SPLINE
SPL {X  -165.650, Y  +484.445, Z    +0.000, E1   +32.277, E3 +483766.169}
SPL {X  -165.650, Y  +481.524, Z    +0.000, E1   +31.089, E3 +483783.620}
SPL {X  -165.650, Y  +478.014, Z    +0.000, E1   +30.826, E3 +483797.227}
SPL {X  -165.650, Y  +474.473, Z    +0.000, E1   +30.943, E3 +483808.552}
SPL {X  -165.650, Y  +470.376, Z    +0.000, E1   +30.888, E3 +483823.081}
SPL {X  -165.650, Y  +465.146, Z    +0.000, E1   +30.883, E3 +483841.012}
SPL {X  -165.650, Y  +461.106, Z    +0.000, E1   +30.916, E3 +483854.430}
SPL {X  -165.650, Y  +458.435, Z    +0.000, E1   +30.759, E3 +483864.638}
SPL {X  -165.650, Y  +454.220, Z    +0.000, E1   +30.954, E3 +483877.871}
SPL {X  -165.650, Y  +450.433, Z    +0.000, E1   +30.789, E3 +483891.835}
SPL {X  -165.650, Y  +447.097, Z    +0.000, E1   +30.843, E3 +483902.884}
SPL {X  -165.650, Y  +443.673, Z    +0.000, E1   +30.907, E3 +483914.192}
SPL {X  -165.650, Y  +440.976, Z    +0.000, E1   +30.719, E3 +483924.648}
SPL {X  -165.650, Y  +436.324, Z    +0.000, E1   +30.994, E3 +483938.935}
SPL {X  -165.650, Y  +432.765, Z    +0.000, E1   +30.831, E3 +483951.935}
SPL {X  -165.650, Y  +429.309, Z    +0.000, E1   +30.920, E3 +483963.276}
SPL {X  -165.650, Y  +424.918, Z    +0.000, E1   +30.862, E3 +483978.733}
SPL {X  -165.650, Y  +421.437, Z    +0.000, E1   +30.833, E3 +483990.701}
SPL {X  -165.650, Y  +418.489, Z    +0.000, E1   +30.835, E3 +484000.818}
SPL {X  -165.650, Y  +414.127, Z    +0.000, E1   +30.869, E3 +484015.726}
SPL {X  -165.650, Y  +408.547, Z    +0.000, E1   +30.964, E3 +484034.142}
SPL {X  -165.650, Y  +405.433, Z    +0.000, E1   +30.730, E3 +484046.119}
SPL {X  -165.650, Y  +402.516, Z    +0.000, E1   +30.874, E3 +484055.242}
SPL {X  -165.650, Y  +398.147, Z    +0.000, E1   +30.902, E3 +484070.120}
SPL {X  -165.650, Y  +394.694, Z    +0.000, E1   +30.805, E3 +484082.429}
SPL {X  -165.650, Y  +391.522, Z    +0.000, E1   +30.837, E3 +484093.110}
SPL {X  -165.650, Y  +387.533, Z    +0.000, E1   +30.858, E3 +484106.736}
SPL {X  -165.650, Y  +383.627, Z    +0.000, E1   +30.885, E3 +484119.796}
SPL {X  -165.650, Y  +379.886, Z    +0.000, E1   +30.887, E3 +484132.684}
SPL {X  -165.614, Y  +375.058, Z    +0.000, E1   +30.905, E3 +484149.137}
SPL {X  -165.492, Y  +371.263, Z    +0.000, E1   +30.913, E3 +484161.851}
SPL {X  -165.379, Y  +369.027, Z    +0.000, E1   +30.727, E3 +484170.790}
SPL {X  -165.167, Y  +365.866, Z    +0.000, E1   +30.741, E3 +484181.564}
SPL {X  -164.892, Y  +362.671, Z    +0.000, E1   +30.830, E3 +484191.888}
SPL {X  -164.570, Y  +359.612, Z    +0.000, E1   +30.773, E3 +484202.700}
SPL {X  -164.104, Y  +355.923, Z    +0.000, E1   +30.626, E3 +484216.417}
SPL {X  -163.573, Y  +352.353, Z    +0.000, E1   +30.451, E3 +484229.682}
SPL {X  -162.476, Y  +346.230, Z    +0.000, E1   +31.677, E3 +484242.263}
SPL {X  -152.976, Y  +314.952, Z    +0.000, E1   +38.607, E3 +484291.228}
SPL {X  -137.967, Y  +286.821, Z    +0.000, E1   +43.969, E3 +484334.449}
ENDSPLINE

SPLINE
SPL {X  -149.143, Y  +306.414, Z    +0.000, E1   +36.361, E3 +484385.581}
SPL {X  -163.091, Y  +349.496, Z    +0.000, E1   +19.699, E3 +484342.364}
SPL {X  -165.027, Y  +364.142, Z    +0.000, E1   +12.054, E3 +484345.505}
SPL {X  -165.612, Y  +374.969, Z    +0.000, E1    +5.630, E3 +484350.687}
SPL {X  -165.650, Y  +383.362, Z    +0.000, E1    +0.177, E3 +484335.306}
SPL {X  -165.650, Y  +383.923, Z    +0.000, E1    -0.215, E3 +484348.463}
SPL {X  -165.650, Y  +388.083, Z    +0.000, E1    -3.355, E3 +484347.327}
SPL {X  -165.650, Y  +393.983, Z    +0.000, E1    -8.501, E3 +484343.725}
SPL {X  -165.650, Y  +402.241, Z    +0.000, E1   -16.711, E3 +484338.237}
SPL {X  -165.650, Y  +414.811, Z    +0.000, E1   -28.314, E3 +484337.767}
SPL {X  -165.650, Y  +423.479, Z    +0.000, E1   -29.012, E3 +484361.696}
SPL {X  -165.650, Y  +441.276, Z    +0.000, E1   -37.343, E3 +484373.385}
SPL {X  -165.650, Y  +462.890, Z    +0.000, E1   -40.484, E3 +484407.468}
ENDSPLINE

SPLINE
SPL {X  -165.650, Y  +446.920, Z    +0.000, E1   -31.238, E3 +484419.794}
ENDSPLINE

SPLINE
SPL {X  -165.650, Y  +447.935, Z    +0.000, E1   -30.213, E3 +484430.081}
SPL {X  -165.650, Y  +451.020, Z    +0.000, E1   -30.224, E3 +484440.902}
SPL {X  -165.650, Y  +454.519, Z    +0.000, E1   -30.374, E3 +484452.084}
SPL {X  -165.650, Y  +456.542, Z    +0.000, E1   -29.986, E3 +484461.829}
SPL {X  -165.650, Y  +460.618, Z    +0.000, E1   -30.298, E3 +484474.149}
SPL {X  -165.650, Y  +463.853, Z    +0.000, E1   -30.103, E3 +484486.750}
SPL {X  -165.650, Y  +468.397, Z    +0.000, E1   -30.302, E3 +484501.554}
SPL {X  -165.650, Y  +472.566, Z    +0.000, E1   -30.124, E3 +484517.263}
SPL {X  -165.650, Y  +475.265, Z    +0.000, E1   -30.034, E3 +484527.301}
SPL {X  -165.650, Y  +479.559, Z    +0.000, E1   -30.258, E3 +484541.165}
SPL {X  -165.650, Y  +484.477, Z    +0.000, E1   -30.274, E3 +484558.174}
SPL {X  -165.650, Y  +488.041, Z    +0.000, E1   -30.253, E3 +484570.730}
SPL {X  -165.650, Y  +491.281, Z    +0.000, E1   -30.148, E3 +484582.868}
SPL {X  -165.650, Y  +495.051, Z    +0.000, E1   -30.213, E3 +484595.676}
SPL {X  -165.650, Y  +498.418, Z    +0.000, E1   -30.282, E3 +484606.969}
SPL {X  -165.650, Y  +502.421, Z    +0.000, E1   -30.263, E3 +484621.327}
SPL {X  -165.650, Y  +506.344, Z    +0.000, E1   -30.129, E3 +484635.856}
SPL {X  -165.650, Y  +509.866, Z    +0.000, E1   -30.236, E3 +484647.526}
SPL {X  -165.650, Y  +513.685, Z    +0.000, E1   -30.234, E3 +484661.022}
SPL {X  -165.650, Y  +517.919, Z    +0.000, E1   -30.227, E3 +484675.929}
SPL {X  -165.650, Y  +522.822, Z    +0.000, E1   -30.289, E3 +484692.818}
SPL {X  -165.650, Y  +527.393, Z    +0.000, E1   -30.104, E3 +484710.066}
SPL {X  -165.650, Y  +531.783, Z    +0.000, E1   -30.416, E3 +484723.244}
SPL {X  -165.650, Y  +534.115, Z    +0.000, E1   -30.089, E3 +484733.626}
SPL {X  -165.650, Y  +537.522, Z    +0.000, E1   -30.251, E3 +484744.540}
SPL {X  -165.650, Y  +540.621, Z    +0.000, E1   -30.014, E3 +484757.101}
SPL {X  -165.650, Y  +544.944, Z    +0.000, E1   -30.447, E3 +484769.301}
SPL {X  -165.650, Y  +548.549, Z    +0.000, E1   -30.216, E3 +484783.624}
SPL {X  -165.650, Y  +553.092, Z    +0.000, E1   -30.157, E3 +484799.967}
SPL {X  -165.650, Y  +556.274, Z    +0.000, E1   -30.127, E3 +484811.221}
SPL {X  -165.650, Y  +560.243, Z    +0.000, E1   -30.214, E3 +484824.887}
SPL {X  -165.650, Y  +565.528, Z    +0.000, E1   -30.192, E3 +484843.579}
SPL {X  -165.650, Y  +570.048, Z    +0.000, E1   -30.238, E3 +484859.010}
SPL {X  -165.650, Y  +573.110, Z    +0.000, E1   -30.057, E3 +484870.995}
SPL {X  -165.650, Y  +576.497, Z    +0.000, E1   -30.234, E3 +484881.693}
SPL {X  -165.650, Y  +580.354, Z    +0.000, E1   -30.196, E3 +484895.709}
SPL {X  -165.650, Y  +585.053, Z    +0.000, E1   -30.090, E3 +484912.944}
ENDSPLINE

SPLINE
SPL {X  -165.650, Y  +484.445, Z    +0.000, E1   +32.277, E3 +484930.348}
SPL {X  -165.650, Y  +481.524, Z    +0.000, E1   +31.089, E3 +484947.799}
SPL {X  -165.650, Y  +478.014, Z    +0.000, E1   +30.826, E3 +484961.407}
SPL {X  -165.650, Y  +474.473, Z    +0.000, E1   +30.943, E3 +484972.731}
SPL {X  -165.650, Y  +470.376, Z    +0.000, E1   +30.888, E3 +484987.260}
SPL {X  -165.650, Y  +465.146, Z    +0.000, E1   +30.883, E3 +485005.191}
SPL {X  -165.650, Y  +461.106, Z    +0.000, E1   +30.916, E3 +485018.609}
SPL {X  -165.650, Y  +458.435, Z    +0.000, E1   +30.759, E3 +485028.817}
SPL {X  -165.650, Y  +454.220, Z    +0.000, E1   +30.954, E3 +485042.050}
SPL {X  -165.650, Y  +450.433, Z    +0.000, E1   +30.789, E3 +485056.015}
SPL {X  -165.650, Y  +447.097, Z    +0.000, E1   +30.843, E3 +485067.063}
SPL {X  -165.650, Y  +443.673, Z    +0.000, E1   +30.907, E3 +485078.371}
SPL {X  -165.650, Y  +440.976, Z    +0.000, E1   +30.719, E3 +485088.827}
SPL {X  -165.650, Y  +436.324, Z    +0.000, E1   +30.994, E3 +485103.114}
SPL {X  -165.650, Y  +432.765, Z    +0.000, E1   +30.831, E3 +485116.114}
SPL {X  -165.650, Y  +429.309, Z    +0.000, E1   +30.920, E3 +485127.455}
SPL {X  -165.650, Y  +424.918, Z    +0.000, E1   +30.862, E3 +485142.912}
SPL {X  -165.650, Y  +421.437, Z    +0.000, E1   +30.833, E3 +485154.880}
SPL {X  -165.650, Y  +418.489, Z    +0.000, E1   +30.835, E3 +485164.997}
SPL {X  -165.650, Y  +415.831, Z    +0.000, E1   +30.847, E3 +485173.960}
SPL {X  -165.650, Y  +412.139, Z    +0.000, E1   +30.870, E3 +485186.670}
SPL {X  -165.650, Y  +406.834, Z    +0.000, E1   +30.919, E3 +485204.499}
SPL {X  -165.650, Y  +401.473, Z    +0.000, E1   +30.933, E3 +485222.747}
SPL {X  -165.650, Y  +396.018, Z    +0.000, E1   +30.861, E3 +485241.931}
SPL {X  -165.650, Y  +391.522, Z    +0.000, E1   +30.837, E3 +485257.289}
SPL {X  -165.650, Y  +387.533, Z    +0.000, E1   +30.858, E3 +485270.915}
SPL {X  -165.650, Y  +383.627, Z    +0.000, E1   +30.885, E3 +485283.975}
SPL {X  -165.650, Y  +380.752, Z    +0.000, E1   +30.927, E3 +485293.489}
SPL {X  -165.648, Y  +377.739, Z    +0.000, E1   +30.835, E3 +485304.498}
SPL {X  -165.594, Y  +374.183, Z    +0.000, E1   +30.878, E3 +485316.335}
SPL {X  -165.429, Y  +369.945, Z    +0.000, E1   +30.850, E3 +485331.210}
SPL {X  -165.167, Y  +365.866, Z    +0.000, E1   +30.741, E3 +485345.743}
SPL {X  -164.892, Y  +362.671, Z    +0.000, E1   +30.830, E3 +485356.067}
SPL {X  -164.570, Y  +359.612, Z    +0.000, E1   +30.773, E3 +485366.880}
SPL {X  -164.104, Y  +355.923, Z    +0.000, E1   +30.626, E3 +485380.596}
SPL {X  -163.573, Y  +352.353, Z    +0.000, E1   +30.451, E3 +485393.861}
SPL {X  -162.976, Y  +348.856, Z    +0.000, E1   +30.757, E3 +485403.785}
SPL {X  -161.497, Y  +341.640, Z    +0.000, E1   +33.276, E3 +485411.062}
SPL {X  -152.976, Y  +314.952, Z    +0.000, E1   +38.607, E3 +485455.407}
SPL {X  -137.967, Y  +286.821, Z    +0.000, E1   +43.969, E3 +485498.628}
ENDSPLINE

SPLINE
SPL {X  -153.316, Y  +315.777, Z    +0.000, E1   +33.140, E3 +485541.255}
SPL {X  -164.446, Y  +358.564, Z    +0.000, E1   +15.149, E3 +485506.466}
SPL {X  -165.510, Y  +371.680, Z    +0.000, E1    +7.684, E3 +485510.522}
SPL {X  -165.628, Y  +375.818, Z    +0.000, E1    +5.016, E3 +485518.451}
SPL {X  -165.650, Y  +383.362, Z    +0.000, E1    +0.177, E3 +485499.485}
SPL {X  -165.650, Y  +383.923, Z    +0.000, E1    -0.215, E3 +485512.642}
SPL {X  -165.650, Y  +388.083, Z    +0.000, E1    -3.355, E3 +485511.506}
SPL {X  -165.650, Y  +395.510, Z    +0.000, E1    -9.810, E3 +485507.632}
SPL {X  -165.650, Y  +403.066, Z    +0.000, E1   -17.886, E3 +485500.465}
SPL {X  -165.650, Y  +414.811, Z    +0.000, E1   -28.314, E3 +485501.946}
SPL {X  -165.650, Y  +423.479, Z    +0.000, E1   -29.012, E3 +485525.875}
SPL {X  -165.650, Y  +435.050, Z    +0.000, E1   -34.610, E3 +485534.209}
SPL {X  -165.650, Y  +446.725, Z    +0.000, E1   -39.593, E3 +485540.471}
SPL {X  -165.650, Y  +462.890, Z    +0.000, E1   -40.484, E3 +485571.647}
ENDSPLINE

SPLINE
SPL {X  -165.650, Y  +446.920, Z    +0.000, E1   -31.238, E3 +485583.973}
ENDSPLINE

SPLINE
SPL {X  -165.650, Y  +447.935, Z    +0.000, E1   -30.213, E3 +485594.261}
SPL {X  -165.650, Y  +451.020, Z    +0.000, E1   -30.224, E3 +485605.081}
SPL {X  -165.650, Y  +454.519, Z    +0.000, E1   -30.374, E3 +485616.263}
SPL {X  -165.650, Y  +457.429, Z    +0.000, E1   -30.029, E3 +485628.965}
SPL {X  -165.650, Y  +461.678, Z    +0.000, E1   -30.426, E3 +485641.090}
SPL {X  -165.650, Y  +463.853, Z    +0.000, E1   -30.103, E3 +485650.929}
SPL {X  -165.650, Y  +468.397, Z    +0.000, E1   -30.302, E3 +485665.733}
SPL {X  -165.650, Y  +472.566, Z    +0.000, E1   -30.124, E3 +485681.442}
SPL {X  -165.650, Y  +476.540, Z    +0.000, E1   -30.193, E3 +485694.987}
SPL {X  -165.650, Y  +480.320, Z    +0.000, E1   -30.163, E3 +485708.464}
SPL {X  -165.650, Y  +484.477, Z    +0.000, E1   -30.274, E3 +485722.354}
SPL {X  -165.650, Y  +488.041, Z    +0.000, E1   -30.253, E3 +485734.909}
SPL {X  -165.650, Y  +491.281, Z    +0.000, E1   -30.148, E3 +485747.047}
SPL {X  -165.650, Y  +495.051, Z    +0.000, E1   -30.213, E3 +485759.855}
SPL {X  -165.650, Y  +498.418, Z    +0.000, E1   -30.282, E3 +485771.148}
SPL {X  -165.650, Y  +500.833, Z    +0.000, E1   -30.191, E3 +485780.197}
SPL {X  -165.650, Y  +504.246, Z    +0.000, E1   -30.231, E3 +485792.064}
SPL {X  -165.650, Y  +507.017, Z    +0.000, E1   -30.108, E3 +485802.472}
SPL {X  -165.650, Y  +510.660, Z    +0.000, E1   -30.223, E3 +485814.739}
SPL {X  -165.650, Y  +514.670, Z    +0.000, E1   -30.278, E3 +485828.249}
SPL {X  -165.650, Y  +517.919, Z    +0.000, E1   -30.227, E3 +485840.108}
SPL {X  -165.650, Y  +521.521, Z    +0.000, E1   -30.210, E3 +485852.783}
SPL {X  -165.650, Y  +525.344, Z    +0.000, E1   -30.269, E3 +485865.889}
SPL {X  -165.650, Y  +528.152, Z    +0.000, E1   -29.991, E3 +485877.530}
SPL {X  -165.650, Y  +531.783, Z    +0.000, E1   -30.416, E3 +485887.423}
SPL {X  -165.650, Y  +534.115, Z    +0.000, E1   -30.089, E3 +485897.805}
SPL {X  -165.650, Y  +537.522, Z    +0.000, E1   -30.251, E3 +485908.719}
SPL {X  -165.650, Y  +540.621, Z    +0.000, E1   -30.014, E3 +485921.280}
SPL {X  -165.650, Y  +544.944, Z    +0.000, E1   -30.447, E3 +485933.480}
SPL {X  -165.650, Y  +547.199, Z    +0.000, E1   -30.132, E3 +485943.453}
SPL {X  -165.650, Y  +550.512, Z    +0.000, E1   -30.197, E3 +485954.779}
SPL {X  -165.650, Y  +553.852, Z    +0.000, E1   -30.156, E3 +485966.720}
SPL {X  -165.650, Y  +557.277, Z    +0.000, E1   -30.150, E3 +485978.894}
SPL {X  -165.650, Y  +561.168, Z    +0.000, E1   -30.194, E3 +485992.276}
SPL {X  -165.650, Y  +564.449, Z    +0.000, E1   -30.167, E3 +486003.959}
SPL {X  -165.650, Y  +566.935, Z    +0.000, E1   -30.135, E3 +486012.865}
SPL {X  -165.650, Y  +570.048, Z    +0.000, E1   -30.238, E3 +486023.190}
SPL {X  -165.650, Y  +573.110, Z    +0.000, E1   -30.057, E3 +486035.175}
SPL {X  -165.650, Y  +576.497, Z    +0.000, E1   -30.234, E3 +486045.872}
SPL {X  -165.650, Y  +578.919, Z    +0.000, E1   -30.237, E3 +486054.318}
SPL {X  -165.650, Y  +582.378, Z    +0.000, E1   -30.208, E3 +486066.901}
SPL {X  -165.650, Y  +585.733, Z    +0.000, E1   -29.896, E3 +486080.661}
ENDSPLINE

SPLINE
SPL {X  -165.650, Y  +484.445, Z    +0.000, E1   +32.277, E3 +486094.528}
SPL {X  -165.650, Y  +481.524, Z    +0.000, E1   +31.089, E3 +486111.978}
SPL {X  -165.650, Y  +478.014, Z    +0.000, E1   +30.826, E3 +486125.586}
SPL {X  -165.650, Y  +474.473, Z    +0.000, E1   +30.943, E3 +486136.910}
SPL {X  -165.650, Y  +471.826, Z    +0.000, E1   +30.770, E3 +486147.094}
SPL {X  -165.650, Y  +467.753, Z    +0.000, E1   +30.878, E3 +486160.467}
SPL {X  -165.650, Y  +463.837, Z    +0.000, E1   +30.924, E3 +486173.401}
SPL {X  -165.650, Y  +461.106, Z    +0.000, E1   +30.916, E3 +486182.788}
SPL {X  -165.650, Y  +458.435, Z    +0.000, E1   +30.759, E3 +486192.996}
SPL {X  -165.650, Y  +454.220, Z    +0.000, E1   +30.954, E3 +486206.229}
SPL {X  -165.650, Y  +450.433, Z    +0.000, E1   +30.789, E3 +486220.194}
SPL {X  -165.650, Y  +447.097, Z    +0.000, E1   +30.843, E3 +486231.242}
SPL {X  -165.650, Y  +443.673, Z    +0.000, E1   +30.907, E3 +486242.550}
SPL {X  -165.650, Y  +440.976, Z    +0.000, E1   +30.719, E3 +486253.006}
SPL {X  -165.650, Y  +436.324, Z    +0.000, E1   +30.994, E3 +486267.293}
SPL {X  -165.650, Y  +432.765, Z    +0.000, E1   +30.831, E3 +486280.293}
SPL {X  -165.650, Y  +429.309, Z    +0.000, E1   +30.920, E3 +486291.634}
SPL {X  -165.650, Y  +424.918, Z    +0.000, E1   +30.862, E3 +486307.091}
SPL {X  -165.650, Y  +421.437, Z    +0.000, E1   +30.833, E3 +486319.059}
SPL {X  -165.650, Y  +417.366, Z    +0.000, E1   +30.879, E3 +486332.900}
SPL {X  -165.650, Y  +412.139, Z    +0.000, E1   +30.870, E3 +486350.849}
SPL {X  -165.650, Y  +406.834, Z    +0.000, E1   +30.919, E3 +486368.678}
SPL {X  -165.650, Y  +402.516, Z    +0.000, E1   +30.874, E3 +486383.600}
SPL {X  -165.650, Y  +398.147, Z    +0.000, E1   +30.902, E3 +486398.479}
SPL {X  -165.650, Y  +394.694, Z    +0.000, E1   +30.805, E3 +486410.787}
SPL {X  -165.650, Y  +391.522, Z    +0.000, E1   +30.837, E3 +486421.468}
SPL {X  -165.650, Y  +387.533, Z    +0.000, E1   +30.858, E3 +486435.094}
SPL {X  -165.650, Y  +383.627, Z    +0.000, E1   +30.885, E3 +486448.154}
SPL {X  -165.650, Y  +380.752, Z    +0.000, E1   +30.927, E3 +486457.668}
SPL {X  -165.648, Y  +377.739, Z    +0.000, E1   +30.835, E3 +486468.678}
SPL {X  -165.594, Y  +374.183, Z    +0.000, E1   +30.878, E3 +486480.514}
SPL {X  -165.492, Y  +371.263, Z    +0.000, E1   +30.913, E3 +486490.209}
SPL {X  -165.379, Y  +369.027, Z    +0.000, E1   +30.727, E3 +486499.148}
SPL {X  -165.167, Y  +365.866, Z    +0.000, E1   +30.741, E3 +486509.922}
SPL {X  -164.892, Y  +362.671, Z    +0.000, E1   +30.830, E3 +486520.246}
SPL {X  -164.570, Y  +359.612, Z    +0.000, E1   +30.773, E3 +486531.059}
SPL {X  -164.104, Y  +355.923, Z    +0.000, E1   +30.626, E3 +486544.775}
SPL {X  -163.573, Y  +352.353, Z    +0.000, E1   +30.451, E3 +486558.040}
SPL {X  -162.476, Y  +346.230, Z    +0.000, E1   +31.677, E3 +486570.621}
SPL {X  -152.976, Y  +314.952, Z    +0.000, E1   +38.607, E3 +486619.586}
SPL {X  -137.967, Y  +286.821, Z    +0.000, E1   +43.969, E3 +486662.807}
ENDSPLINE

SPLINE
SPL {X  -153.316, Y  +315.777, Z    +0.000, E1   +33.140, E3 +486705.435}
SPL {X  -164.446, Y  +358.564, Z    +0.000, E1   +15.149, E3 +486670.645}
SPL {X  -165.379, Y  +369.025, Z    +0.000, E1    +9.158, E3 +486676.370}
SPL {X  -165.612, Y  +374.969, Z    +0.000, E1    +5.630, E3 +486679.046}
SPL {X  -165.650, Y  +383.362, Z    +0.000, E1    +0.177, E3 +486663.664}
SPL {X  -165.650, Y  +383.923, Z    +0.000, E1    -0.215, E3 +486676.821}
SPL {X  -165.650, Y  +388.083, Z    +0.000, E1    -3.355, E3 +486675.685}
SPL {X  -165.650, Y  +393.983, Z    +0.000, E1    -8.501, E3 +486672.083}
SPL {X  -165.650, Y  +402.241, Z    +0.000, E1   -16.711, E3 +486666.595}
SPL {X  -165.650, Y  +416.345, Z    +0.000, E1   -29.511, E3 +486666.387}
SPL {X  -165.650, Y  +422.331, Z    +0.000, E1   -27.760, E3 +486691.886}
SPL {X  -165.650, Y  +441.276, Z    +0.000, E1   -37.343, E3 +486701.743}
SPL {X  -165.650, Y  +462.890, Z    +0.000, E1   -40.484, E3 +486735.826}
ENDSPLINE

SPLINE
SPL {X  -165.650, Y  +446.920, Z    +0.000, E1   -31.238, E3 +486748.152}
ENDSPLINE

SPLINE
SPL {X  -165.650, Y  +447.935, Z    +0.000, E1   -30.213, E3 +486758.440}
SPL {X  -165.650, Y  +451.020, Z    +0.000, E1   -30.224, E3 +486769.260}
SPL {X  -165.650, Y  +454.519, Z    +0.000, E1   -30.374, E3 +486780.442}
SPL {X  -165.650, Y  +457.429, Z    +0.000, E1   -30.029, E3 +486793.144}
SPL {X  -165.650, Y  +461.678, Z    +0.000, E1   -30.426, E3 +486805.269}
SPL {X  -165.650, Y  +463.853, Z    +0.000, E1   -30.103, E3 +486815.108}
SPL {X  -165.650, Y  +468.397, Z    +0.000, E1   -30.302, E3 +486829.912}
SPL {X  -165.650, Y  +472.566, Z    +0.000, E1   -30.124, E3 +486845.622}
SPL {X  -165.650, Y  +476.540, Z    +0.000, E1   -30.193, E3 +486859.166}
SPL {X  -165.650, Y  +481.042, Z    +0.000, E1   -30.192, E3 +486875.111}
SPL {X  -165.650, Y  +485.236, Z    +0.000, E1   -30.294, E3 +486888.966}
SPL {X  -165.650, Y  +489.057, Z    +0.000, E1   -30.341, E3 +486902.172}
SPL {X  -165.650, Y  +491.647, Z    +0.000, E1   -29.894, E3 +486914.106}
SPL {X  -165.650, Y  +495.051, Z    +0.000, E1   -30.213, E3 +486924.035}
SPL {X  -165.650, Y  +498.418, Z    +0.000, E1   -30.282, E3 +486935.327}
SPL {X  -165.650, Y  +502.421, Z    +0.000, E1   -30.263, E3 +486949.685}
SPL {X  -165.650, Y  +506.344, Z    +0.000, E1   -30.129, E3 +486964.214}
SPL {X  -165.650, Y  +509.866, Z    +0.000, E1   -30.236, E3 +486975.884}
SPL {X  -165.650, Y  +513.685, Z    +0.000, E1   -30.234, E3 +486989.380}
SPL {X  -165.650, Y  +517.919, Z    +0.000, E1   -30.227, E3 +487004.287}
SPL {X  -165.650, Y  +521.521, Z    +0.000, E1   -30.210, E3 +487016.962}
SPL {X  -165.650, Y  +525.344, Z    +0.000, E1   -30.269, E3 +487030.068}
SPL {X  -165.650, Y  +528.152, Z    +0.000, E1   -29.991, E3 +487041.709}
SPL {X  -165.650, Y  +531.783, Z    +0.000, E1   -30.416, E3 +487051.602}
SPL {X  -165.650, Y  +534.115, Z    +0.000, E1   -30.089, E3 +487061.984}
SPL {X  -165.650, Y  +537.522, Z    +0.000, E1   -30.251, E3 +487072.898}
SPL {X  -165.650, Y  +540.621, Z    +0.000, E1   -30.014, E3 +487085.459}
SPL {X  -165.650, Y  +544.944, Z    +0.000, E1   -30.447, E3 +487097.659}
SPL {X  -165.650, Y  +548.549, Z    +0.000, E1   -30.216, E3 +487111.982}
SPL {X  -165.650, Y  +553.092, Z    +0.000, E1   -30.157, E3 +487128.325}
SPL {X  -165.650, Y  +556.274, Z    +0.000, E1   -30.127, E3 +487139.579}
SPL {X  -165.650, Y  +560.243, Z    +0.000, E1   -30.214, E3 +487153.245}
SPL {X  -165.650, Y  +565.528, Z    +0.000, E1   -30.192, E3 +487171.938}
SPL {X  -165.650, Y  +570.048, Z    +0.000, E1   -30.238, E3 +487187.369}
SPL {X  -165.650, Y  +573.110, Z    +0.000, E1   -30.057, E3 +487199.354}
SPL {X  -165.650, Y  +577.587, Z    +0.000, E1   -30.270, E3 +487213.793}
SPL {X  -165.650, Y  +581.190, Z    +0.000, E1   -30.107, E3 +487227.432}
SPL {X  -165.650, Y  +585.053, Z    +0.000, E1   -30.090, E3 +487241.302}
ENDSPLINE

SPLINE
SPL {X  -165.650, Y  +484.445, Z    +0.000, E1   +32.277, E3 +487258.707}
SPL {X  -165.650, Y  +481.524, Z    +0.000, E1   +31.089, E3 +487276.157}
SPL {X  -165.650, Y  +478.014, Z    +0.000, E1   +30.826, E3 +487289.765}
SPL {X  -165.650, Y  +474.473, Z    +0.000, E1   +30.943, E3 +487301.089}
SPL {X  -165.650, Y  +471.826, Z    +0.000, E1   +30.770, E3 +487311.273}
SPL {X  -165.650, Y  +467.753, Z    +0.000, E1   +30.878, E3 +487324.646}
SPL {X  -165.650, Y  +463.837, Z    +0.000, E1   +30.924, E3 +487337.580}
SPL {X  -165.650, Y  +461.106, Z    +0.000, E1   +30.916, E3 +487346.967}
SPL {X  -165.650, Y  +458.435, Z    +0.000, E1   +30.759, E3 +487357.175}
SPL {X  -165.650, Y  +454.220, Z    +0.000, E1   +30.954, E3 +487370.408}
SPL {X  -165.650, Y  +450.433, Z    +0.000, E1   +30.789, E3 +487384.373}
SPL {X  -165.650, Y  +447.097, Z    +0.000, E1   +30.843, E3 +487395.421}
SPL {X  -165.650, Y  +443.673, Z    +0.000, E1   +30.907, E3 +487406.729}
SPL {X  -165.650, Y  +440.976, Z    +0.000, E1   +30.719, E3 +487417.186}
SPL {X  -165.650, Y  +436.324, Z    +0.000, E1   +30.994, E3 +487431.472}
SPL {X  -165.650, Y  +432.765, Z    +0.000, E1   +30.831, E3 +487444.472}
SPL {X  -165.650, Y  +429.309, Z    +0.000, E1   +30.920, E3 +487455.813}
SPL {X  -165.650, Y  +424.918, Z    +0.000, E1   +30.862, E3 +487471.270}
SPL {X  -165.650, Y  +421.437, Z    +0.000, E1   +30.833, E3 +487483.238}
SPL {X  -165.650, Y  +417.366, Z    +0.000, E1   +30.879, E3 +487497.079}
SPL {X  -165.650, Y  +413.181, Z    +0.000, E1   +30.815, E3 +487511.676}
SPL {X  -165.650, Y  +408.547, Z    +0.000, E1   +30.964, E3 +487526.679}
SPL {X  -165.650, Y  +403.421, Z    +0.000, E1   +30.863, E3 +487544.897}
SPL {X  -165.650, Y  +398.147, Z    +0.000, E1   +30.902, E3 +487562.658}
SPL {X  -165.650, Y  +394.694, Z    +0.000, E1   +30.805, E3 +487574.966}
SPL {X  -165.650, Y  +391.522, Z    +0.000, E1   +30.837, E3 +487585.647}
SPL {X  -165.650, Y  +387.533, Z    +0.000, E1   +30.858, E3 +487599.273}
SPL {X  -165.650, Y  +383.627, Z    +0.000, E1   +30.885, E3 +487612.333}
SPL {X  -165.650, Y  +379.886, Z    +0.000, E1   +30.887, E3 +487625.222}
SPL {X  -165.614, Y  +375.058, Z    +0.000, E1   +30.905, E3 +487641.675}
SPL {X  -165.492, Y  +371.263, Z    +0.000, E1   +30.913, E3 +487654.389}
SPL {X  -165.379, Y  +369.027, Z    +0.000, E1   +30.727, E3 +487663.327}
SPL {X  -165.167, Y  +365.866, Z    +0.000, E1   +30.741, E3 +487674.101}
SPL {X  -164.892, Y  +362.671, Z    +0.000, E1   +30.830, E3 +487684.425}
SPL {X  -164.570, Y  +359.612, Z    +0.000, E1   +30.773, E3 +487695.238}
SPL {X  -164.104, Y  +355.923, Z    +0.000, E1   +30.626, E3 +487708.954}
SPL {X  -163.573, Y  +352.353, Z    +0.000, E1   +30.451, E3 +487722.219}
SPL {X  -162.476, Y  +346.230, Z    +0.000, E1   +31.677, E3 +487734.800}
SPL {X  -152.976, Y  +314.952, Z    +0.000, E1   +38.607, E3 +487783.765}
SPL {X  -137.967, Y  +286.821, Z    +0.000, E1   +43.969, E3 +487826.986}
ENDSPLINE

SPLINE
SPL {X  -153.316, Y  +315.777, Z    +0.000, E1   +33.140, E3 +487869.614}
SPL {X  -164.446, Y  +358.564, Z    +0.000, E1   +15.149, E3 +487834.825}
SPL {X  -165.510, Y  +371.680, Z    +0.000, E1    +7.684, E3 +487838.880}
SPL {X  -165.628, Y  +375.818, Z    +0.000, E1    +5.016, E3 +487846.810}
SPL {X  -165.650, Y  +383.362, Z    +0.000, E1    +0.177, E3 +487827.843}
SPL {X  -165.650, Y  +383.923, Z    +0.000, E1    -0.215, E3 +487841.001}
SPL {X  -165.650, Y  +388.083, Z    +0.000, E1    -3.355, E3 +487839.864}
SPL {X  -165.650, Y  +393.983, Z    +0.000, E1    -8.501, E3 +487836.262}
SPL {X  -165.650, Y  +402.241, Z    +0.000, E1   -16.711, E3 +487830.774}
SPL {X  -165.650, Y  +414.811, Z    +0.000, E1   -28.314, E3 +487830.305}
SPL {X  -165.650, Y  +423.479, Z    +0.000, E1   -29.012, E3 +487854.233}
SPL {X  -165.650, Y  +441.276, Z    +0.000, E1   -37.343, E3 +487865.922}
SPL {X  -165.650, Y  +462.890, Z    +0.000, E1   -40.484, E3 +487900.005}
ENDSPLINE

SPLINE
SPL {X  -165.650, Y  +446.920, Z    +0.000, E1   -31.238, E3 +487912.331}
ENDSPLINE

SPLINE
SPL {X  -165.650, Y  +447.935, Z    +0.000, E1   -30.213, E3 +487922.619}
SPL {X  -165.650, Y  +451.020, Z    +0.000, E1   -30.224, E3 +487933.439}
SPL {X  -165.650, Y  +454.519, Z    +0.000, E1   -30.374, E3 +487944.621}
SPL {X  -165.650, Y  +456.542, Z    +0.000, E1   -29.986, E3 +487954.366}
SPL {X  -165.650, Y  +460.618, Z    +0.000, E1   -30.298, E3 +487966.687}
SPL {X  -165.650, Y  +463.853, Z    +0.000, E1   -30.103, E3 +487979.288}
SPL {X  -165.650, Y  +468.397, Z    +0.000, E1   -30.302, E3 +487994.091}
SPL {X  -165.650, Y  +472.566, Z    +0.000, E1   -30.124, E3 +488009.801}
SPL {X  -165.650, Y  +475.265, Z    +0.000, E1   -30.034, E3 +488019.838}
SPL {X  -165.650, Y  +477.862, Z    +0.000, E1   -30.319, E3 +488027.030}
SPL {X  -165.650, Y  +481.042, Z    +0.000, E1   -30.192, E3 +488039.290}
SPL {X  -165.650, Y  +485.236, Z    +0.000, E1   -30.294, E3 +488053.146}
SPL {X  -165.650, Y  +488.041, Z    +0.000, E1   -30.253, E3 +488063.267}
SPL {X  -165.650, Y  +491.281, Z    +0.000, E1   -30.148, E3 +488075.405}
SPL {X  -165.650, Y  +495.051, Z    +0.000, E1   -30.213, E3 +488088.214}
SPL {X  -165.650, Y  +499.546, Z    +0.000, E1   -30.283, E3 +488103.656}
SPL {X  -165.650, Y  +503.544, Z    +0.000, E1   -30.247, E3 +488117.725}
SPL {X  -165.650, Y  +506.344, Z    +0.000, E1   -30.129, E3 +488128.394}
SPL {X  -165.650, Y  +510.660, Z    +0.000, E1   -30.223, E3 +488143.097}
SPL {X  -165.650, Y  +514.670, Z    +0.000, E1   -30.278, E3 +488156.607}
SPL {X  -165.650, Y  +517.919, Z    +0.000, E1   -30.227, E3 +488168.466}
SPL {X  -165.650, Y  +521.521, Z    +0.000, E1   -30.210, E3 +488181.141}
SPL {X  -165.650, Y  +525.344, Z    +0.000, E1   -30.269, E3 +488194.247}
SPL {X  -165.650, Y  +528.152, Z    +0.000, E1   -29.991, E3 +488205.888}
SPL {X  -165.650, Y  +531.783, Z    +0.000, E1   -30.416, E3 +488215.781}
SPL {X  -165.650, Y  +534.115, Z    +0.000, E1   -30.089, E3 +488226.163}
SPL {X  -165.650, Y  +537.522, Z    +0.000, E1   -30.251, E3 +488237.077}
SPL {X  -165.650, Y  +540.621, Z    +0.000, E1   -30.014, E3 +488249.638}
SPL {X  -165.650, Y  +544.944, Z    +0.000, E1   -30.447, E3 +488261.838}
SPL {X  -165.650, Y  +547.199, Z    +0.000, E1   -30.132, E3 +488271.811}
SPL {X  -165.650, Y  +550.512, Z    +0.000, E1   -30.197, E3 +488283.137}
SPL {X  -165.650, Y  +553.852, Z    +0.000, E1   -30.156, E3 +488295.078}
SPL {X  -165.650, Y  +557.277, Z    +0.000, E1   -30.150, E3 +488307.252}
SPL {X  -165.650, Y  +561.168, Z    +0.000, E1   -30.194, E3 +488320.634}
SPL {X  -165.650, Y  +564.449, Z    +0.000, E1   -30.167, E3 +488332.317}
SPL {X  -165.650, Y  +566.935, Z    +0.000, E1   -30.135, E3 +488341.223}
SPL {X  -165.650, Y  +570.048, Z    +0.000, E1   -30.238, E3 +488351.548}
SPL {X  -165.650, Y  +573.110, Z    +0.000, E1   -30.057, E3 +488363.533}
SPL {X  -165.650, Y  +577.587, Z    +0.000, E1   -30.270, E3 +488377.972}
SPL {X  -165.650, Y  +581.190, Z    +0.000, E1   -30.107, E3 +488391.611}
SPL {X  -165.650, Y  +585.053, Z    +0.000, E1   -30.090, E3 +488405.481}
ENDSPLINE

SPLINE
SPL {X  -165.650, Y  +484.445, Z    +0.000, E1   +32.277, E3 +488422.886}
SPL {X  -165.650, Y  +481.524, Z    +0.000, E1   +31.089, E3 +488440.336}
SPL {X  -165.650, Y  +478.014, Z    +0.000, E1   +30.826, E3 +488453.944}
SPL {X  -165.650, Y  +474.473, Z    +0.000, E1   +30.943, E3 +488465.268}
SPL {X  -165.650, Y  +471.826, Z    +0.000, E1   +30.770, E3 +488475.452}
SPL {X  -165.650, Y  +467.753, Z    +0.000, E1   +30.878, E3 +488488.825}
SPL {X  -165.650, Y  +463.837, Z    +0.000, E1   +30.924, E3 +488501.759}
SPL {X  -165.650, Y  +461.106, Z    +0.000, E1   +30.916, E3 +488511.146}
SPL {X  -165.650, Y  +458.435, Z    +0.000, E1   +30.759, E3 +488521.354}
SPL {X  -165.650, Y  +454.220, Z    +0.000, E1   +30.954, E3 +488534.587}
SPL {X  -165.650, Y  +450.433, Z    +0.000, E1   +30.789, E3 +488548.552}
SPL {X  -165.650, Y  +447.097, Z    +0.000, E1   +30.843, E3 +488559.601}
SPL {X  -165.650, Y  +443.673, Z    +0.000, E1   +30.907, E3 +488570.908}
SPL {X  -165.650, Y  +439.486, Z    +0.000, E1   +30.857, E3 +488585.717}
SPL {X  -165.650, Y  +435.146, Z    +0.000, E1   +30.969, E3 +488599.637}
SPL {X  -165.650, Y  +431.607, Z    +0.000, E1   +30.889, E3 +488612.351}
SPL {X  -165.650, Y  +427.340, Z    +0.000, E1   +30.870, E3 +488627.063}
SPL {X  -165.650, Y  +423.901, Z    +0.000, E1   +30.858, E3 +488638.819}
SPL {X  -165.650, Y  +421.437, Z    +0.000, E1   +30.833, E3 +488647.418}
SPL {X  -165.650, Y  +418.489, Z    +0.000, E1   +30.835, E3 +488657.534}
SPL {X  -165.650, Y  +414.127, Z    +0.000, E1   +30.869, E3 +488672.443}
SPL {X  -165.650, Y  +408.547, Z    +0.000, E1   +30.964, E3 +488690.858}
SPL {X  -165.650, Y  +405.433, Z    +0.000, E1   +30.730, E3 +488702.836}
SPL {X  -165.650, Y  +402.516, Z    +0.000, E1   +30.874, E3 +488711.958}
SPL {X  -165.650, Y  +398.147, Z    +0.000, E1   +30.902, E3 +488726.837}
SPL {X  -165.650, Y  +394.694, Z    +0.000, E1   +30.805, E3 +488739.145}
SPL {X  -165.650, Y  +391.522, Z    +0.000, E1   +30.837, E3 +488749.826}
SPL {X  -165.650, Y  +387.533, Z    +0.000, E1   +30.858, E3 +488763.452}
SPL {X  -165.650, Y  +383.627, Z    +0.000, E1   +30.885, E3 +488776.512}
SPL {X  -165.650, Y  +380.752, Z    +0.000, E1   +30.927, E3 +488786.026}
SPL {X  -165.648, Y  +377.739, Z    +0.000, E1   +30.835, E3 +488797.036}
SPL {X  -165.594, Y  +374.183, Z    +0.000, E1   +30.878, E3 +488808.873}
SPL {X  -165.429, Y  +369.945, Z    +0.000, E1   +30.850, E3 +488823.748}
SPL {X  -165.167, Y  +365.866, Z    +0.000, E1   +30.741, E3 +488838.280}
SPL {X  -164.892, Y  +362.671, Z    +0.000, E1   +30.830, E3 +488848.604}
SPL {X  -164.570, Y  +359.612, Z    +0.000, E1   +30.773, E3 +488859.417}
SPL {X  -164.104, Y  +355.923, Z    +0.000, E1   +30.626, E3 +488873.133}
SPL {X  -163.573, Y  +352.353, Z    +0.000, E1   +30.451, E3 +488886.398}
SPL {X  -162.976, Y  +348.856, Z    +0.000, E1   +30.757, E3 +488896.322}
SPL {X  -161.497, Y  +341.640, Z    +0.000, E1   +33.276, E3 +488903.599}
SPL {X  -152.976, Y  +314.952, Z    +0.000, E1   +38.607, E3 +488947.944}
SPL {X  -137.967, Y  +286.821, Z    +0.000, E1   +43.969, E3 +488991.165}
ENDSPLINE

SPLINE
SPL {X  -149.143, Y  +306.414, Z    +0.000, E1   +36.361, E3 +489042.298}
SPL {X  -163.091, Y  +349.496, Z    +0.000, E1   +19.699, E3 +488999.081}
SPL {X  -165.027, Y  +364.142, Z    +0.000, E1   +12.054, E3 +489002.221}
SPL {X  -165.612, Y  +374.969, Z    +0.000, E1    +5.630, E3 +489007.404}
SPL {X  -165.650, Y  +383.362, Z    +0.000, E1    +0.177, E3 +488992.022}
SPL {X  -165.650, Y  +383.923, Z    +0.000, E1    -0.215, E3 +489005.180}
SPL {X  -165.650, Y  +388.083, Z    +0.000, E1    -3.355, E3 +489004.043}
SPL {X  -165.650, Y  +395.510, Z    +0.000, E1    -9.810, E3 +489000.169}
SPL {X  -165.650, Y  +403.066, Z    +0.000, E1   -17.886, E3 +488993.002}
SPL {X  -165.650, Y  +414.811, Z    +0.000, E1   -28.314, E3 +488994.484}
SPL {X  -165.650, Y  +423.479, Z    +0.000, E1   -29.012, E3 +489018.412}
SPL {X  -165.650, Y  +441.276, Z    +0.000, E1   -37.343, E3 +489030.101}
SPL {X  -165.650, Y  +462.890, Z    +0.000, E1   -40.484, E3 +489064.184}
ENDSPLINE

SPLINE
SPL {X  -165.650, Y  +446.920, Z    +0.000, E1   -31.238, E3 +489076.510}
ENDSPLINE

SPLINE
SPL {X  -165.650, Y  +447.935, Z    +0.000, E1   -30.213, E3 +489086.798}
SPL {X  -165.650, Y  +451.020, Z    +0.000, E1   -30.224, E3 +489097.618}
SPL {X  -165.650, Y  +454.519, Z    +0.000, E1   -30.374, E3 +489108.801}
SPL {X  -165.650, Y  +456.542, Z    +0.000, E1   -29.986, E3 +489118.545}
SPL {X  -165.650, Y  +460.618, Z    +0.000, E1   -30.298, E3 +489130.866}
SPL {X  -165.650, Y  +463.853, Z    +0.000, E1   -30.103, E3 +489143.467}
SPL {X  -165.650, Y  +468.397, Z    +0.000, E1   -30.302, E3 +489158.270}
SPL {X  -165.650, Y  +472.566, Z    +0.000, E1   -30.124, E3 +489173.980}
SPL {X  -165.650, Y  +475.265, Z    +0.000, E1   -30.034, E3 +489184.017}
SPL {X  -165.650, Y  +479.559, Z    +0.000, E1   -30.258, E3 +489197.882}
SPL {X  -165.650, Y  +484.477, Z    +0.000, E1   -30.274, E3 +489214.891}
SPL {X  -165.650, Y  +488.041, Z    +0.000, E1   -30.253, E3 +489227.446}
SPL {X  -165.650, Y  +491.281, Z    +0.000, E1   -30.148, E3 +489239.584}
SPL {X  -165.650, Y  +495.051, Z    +0.000, E1   -30.213, E3 +489252.393}
SPL {X  -165.650, Y  +499.546, Z    +0.000, E1   -30.283, E3 +489267.836}
SPL {X  -165.650, Y  +503.544, Z    +0.000, E1   -30.247, E3 +489281.904}
SPL {X  -165.650, Y  +506.344, Z    +0.000, E1   -30.129, E3 +489292.573}
SPL {X  -165.650, Y  +509.866, Z    +0.000, E1   -30.236, E3 +489304.242}
SPL {X  -165.650, Y  +513.685, Z    +0.000, E1   -30.234, E3 +489317.738}
SPL {X  -165.650, Y  +517.919, Z    +0.000, E1   -30.227, E3 +489332.645}
SPL {X  -165.650, Y  +521.521, Z    +0.000, E1   -30.210, E3 +489345.320}
SPL {X  -165.650, Y  +525.344, Z    +0.000, E1   -30.269, E3 +489358.426}
SPL {X  -165.650, Y  +528.152, Z    +0.000, E1   -29.991, E3 +489370.067}
SPL {X  -165.650, Y  +531.783, Z    +0.000, E1   -30.416, E3 +489379.960}
SPL {X  -165.650, Y  +534.115, Z    +0.000, E1   -30.089, E3 +489390.342}
SPL {X  -165.650, Y  +537.522, Z    +0.000, E1   -30.251, E3 +489401.256}
SPL {X  -165.650, Y  +540.621, Z    +0.000, E1   -30.014, E3 +489413.817}
SPL {X  -165.650, Y  +544.944, Z    +0.000, E1   -30.447, E3 +489426.017}
SPL {X  -165.650, Y  +547.199, Z    +0.000, E1   -30.132, E3 +489435.991}
SPL {X  -165.650, Y  +550.512, Z    +0.000, E1   -30.197, E3 +489447.316}
SPL {X  -165.650, Y  +553.852, Z    +0.000, E1   -30.156, E3 +489459.257}
SPL {X  -165.650, Y  +557.277, Z    +0.000, E1   -30.150, E3 +489471.432}
SPL {X  -165.650, Y  +561.168, Z    +0.000, E1   -30.194, E3 +489484.813}
SPL {X  -165.650, Y  +565.528, Z    +0.000, E1   -30.192, E3 +489500.296}
SPL {X  -165.650, Y  +570.048, Z    +0.000, E1   -30.238, E3 +489515.727}
SPL {X  -165.650, Y  +573.110, Z    +0.000, E1   -30.057, E3 +489527.712}
SPL {X  -165.650, Y  +577.587, Z    +0.000, E1   -30.270, E3 +489542.151}
SPL {X  -165.650, Y  +581.190, Z    +0.000, E1   -30.107, E3 +489555.790}
SPL {X  -165.650, Y  +585.053, Z    +0.000, E1   -30.090, E3 +489569.660}
ENDSPLINE

SPLINE
SPL {X  -165.650, Y  +484.445, Z    +0.000, E1   +32.277, E3 +489587.065}
SPL {X  -165.650, Y  +481.524, Z    +0.000, E1   +31.089, E3 +489604.515}
SPL {X  -165.650, Y  +478.014, Z    +0.000, E1   +30.826, E3 +489618.123}
SPL {X  -165.650, Y  +474.473, Z    +0.000, E1   +30.943, E3 +489629.447}
SPL {X  -165.650, Y  +471.826, Z    +0.000, E1   +30.770, E3 +489639.631}
SPL {X  -165.650, Y  +467.753, Z    +0.000, E1   +30.878, E3 +489653.004}
SPL {X  -165.650, Y  +463.837, Z    +0.000, E1   +30.924, E3 +489665.938}
SPL {X  -165.650, Y  +461.106, Z    +0.000, E1   +30.916, E3 +489675.325}
SPL {X  -165.650, Y  +457.156, Z    +0.000, E1   +30.860, E3 +489689.402}
SPL {X  -165.650, Y  +453.156, Z    +0.000, E1   +30.934, E3 +489702.376}
SPL {X  -165.650, Y  +450.433, Z    +0.000, E1   +30.789, E3 +489712.731}
SPL {X  -165.650, Y  +447.097, Z    +0.000, E1   +30.843, E3 +489723.780}
SPL {X  -165.650, Y  +443.673, Z    +0.000, E1   +30.907, E3 +489735.087}
SPL {X  -165.650, Y  +439.486, Z    +0.000, E1   +30.857, E3 +489749.896}
SPL {X  -165.650, Y  +435.146, Z    +0.000, E1   +30.969, E3 +489763.816}
SPL {X  -165.650, Y  +432.765, Z    +0.000, E1   +30.831, E3 +489772.830}
SPL {X  -165.650, Y  +429.309, Z    +0.000, E1   +30.920, E3 +489784.171}
SPL {X  -165.650, Y  +424.918, Z    +0.000, E1   +30.862, E3 +489799.628}
SPL {X  -165.650, Y  +421.437, Z    +0.000, E1   +30.833, E3 +489811.597}
SPL {X  -165.650, Y  +417.366, Z    +0.000, E1   +30.879, E3 +489825.437}
SPL {X  -165.650, Y  +413.181, Z    +0.000, E1   +30.815, E3 +489840.035}
SPL {X  -165.650, Y  +408.547, Z    +0.000, E1   +30.964, E3 +489855.037}
SPL {X  -165.650, Y  +405.433, Z    +0.000, E1   +30.730, E3 +489867.015}
SPL {X  -165.650, Y  +402.516, Z    +0.000, E1   +30.874, E3 +489876.137}
SPL {X  -165.650, Y  +398.147, Z    +0.000, E1   +30.902, E3 +489891.016}
SPL {X  -165.650, Y  +394.694, Z    +0.000, E1   +30.805, E3 +489903.324}
SPL {X  -165.650, Y  +391.522, Z    +0.000, E1   +30.837, E3 +489914.005}
SPL {X  -165.650, Y  +387.533, Z    +0.000, E1   +30.858, E3 +489927.631}
SPL {X  -165.650, Y  +383.627, Z    +0.000, E1   +30.885, E3 +489940.692}
SPL {X  -165.650, Y  +380.752, Z    +0.000, E1   +30.927, E3 +489950.205}
SPL {X  -165.648, Y  +377.739, Z    +0.000, E1   +30.835, E3 +489961.215}
SPL {X  -165.594, Y  +374.183, Z    +0.000, E1   +30.878, E3 +489973.052}
SPL {X  -165.429, Y  +369.945, Z    +0.000, E1   +30.850, E3 +489987.927}
SPL {X  -165.167, Y  +365.866, Z    +0.000, E1   +30.741, E3 +490002.459}
SPL {X  -164.892, Y  +362.671, Z    +0.000, E1   +30.830, E3 +490012.783}
SPL {X  -164.570, Y  +359.612, Z    +0.000, E1   +30.773, E3 +490023.596}
SPL {X  -164.104, Y  +355.923, Z    +0.000, E1   +30.626, E3 +490037.313}
SPL {X  -163.573, Y  +352.353, Z    +0.000, E1   +30.451, E3 +490050.577}
SPL {X  -162.476, Y  +346.230, Z    +0.000, E1   +31.677, E3 +490063.158}
SPL {X  -152.976, Y  +314.952, Z    +0.000, E1   +38.607, E3 +490112.123}
SPL {X  -137.967, Y  +286.821, Z    +0.000, E1   +43.969, E3 +490155.344}
ENDSPLINE

SPLINE
SPL {X  -149.143, Y  +306.414, Z    +0.000, E1   +36.361, E3 +490206.477}
SPL {X  -164.268, Y  +357.145, Z    +0.000, E1   +15.880, E3 +490164.236}
SPL {X  -165.379, Y  +369.025, Z    +0.000, E1    +9.158, E3 +490168.907}
SPL {X  -165.612, Y  +374.969, Z    +0.000, E1    +5.630, E3 +490171.583}
SPL {X  -165.650, Y  +383.362, Z    +0.000, E1    +0.177, E3 +490156.201}
SPL {X  -165.650, Y  +383.923, Z    +0.000, E1    -0.215, E3 +490169.359}
SPL {X  -165.650, Y  +388.083, Z    +0.000, E1    -3.355, E3 +490168.222}
SPL {X  -165.650, Y  +393.983, Z    +0.000, E1    -8.501, E3 +490164.621}
SPL {X  -165.650, Y  +402.241, Z    +0.000, E1   -16.711, E3 +490159.132}
SPL {X  -165.650, Y  +416.345, Z    +0.000, E1   -29.511, E3 +490158.924}
SPL {X  -165.650, Y  +422.331, Z    +0.000, E1   -27.760, E3 +490184.423}
SPL {X  -165.650, Y  +441.276, Z    +0.000, E1   -37.343, E3 +490194.280}
SPL {X  -165.650, Y  +462.890, Z    +0.000, E1   -40.484, E3 +490228.363}
ENDSPLINE

SPLINE
SPL {X  -165.650, Y  +446.920, Z    +0.000, E1   -31.238, E3 +490240.689}
ENDSPLINE

SPLINE
SPL {X  -165.650, Y  +447.935, Z    +0.000, E1   -30.213, E3 +490250.977}
SPL {X  -165.650, Y  +451.020, Z    +0.000, E1   -30.224, E3 +490261.797}
SPL {X  -165.650, Y  +454.519, Z    +0.000, E1   -30.374, E3 +490272.980}
SPL {X  -165.650, Y  +457.429, Z    +0.000, E1   -30.029, E3 +490285.681}
SPL {X  -165.650, Y  +461.678, Z    +0.000, E1   -30.426, E3 +490297.806}
SPL {X  -165.650, Y  +463.853, Z    +0.000, E1   -30.103, E3 +490307.646}
SPL {X  -165.650, Y  +468.397, Z    +0.000, E1   -30.302, E3 +490322.450}
SPL {X  -165.650, Y  +472.566, Z    +0.000, E1   -30.124, E3 +490338.159}
SPL {X  -165.650, Y  +475.265, Z    +0.000, E1   -30.034, E3 +490348.196}
SPL {X  -165.650, Y  +477.862, Z    +0.000, E1   -30.319, E3 +490355.388}
SPL {X  -165.650, Y  +481.042, Z    +0.000, E1   -30.192, E3 +490367.648}
SPL {X  -165.650, Y  +485.236, Z    +0.000, E1   -30.294, E3 +490381.504}
SPL {X  -165.650, Y  +488.041, Z    +0.000, E1   -30.253, E3 +490391.625}
SPL {X  -165.650, Y  +491.281, Z    +0.000, E1   -30.148, E3 +490403.763}
SPL {X  -165.650, Y  +495.051, Z    +0.000, E1   -30.213, E3 +490416.572}
SPL {X  -165.650, Y  +499.546, Z    +0.000, E1   -30.283, E3 +490432.015}
SPL {X  -165.650, Y  +503.544, Z    +0.000, E1   -30.247, E3 +490446.083}
SPL {X  -165.650, Y  +506.344, Z    +0.000, E1   -30.129, E3 +490456.752}
SPL {X  -165.650, Y  +509.866, Z    +0.000, E1   -30.236, E3 +490468.421}
SPL {X  -165.650, Y  +513.685, Z    +0.000, E1   -30.234, E3 +490481.918}
SPL {X  -165.650, Y  +517.919, Z    +0.000, E1   -30.227, E3 +490496.824}
SPL {X  -165.650, Y  +521.521, Z    +0.000, E1   -30.210, E3 +490509.499}
SPL {X  -165.650, Y  +525.344, Z    +0.000, E1   -30.269, E3 +490522.605}
SPL {X  -165.650, Y  +528.152, Z    +0.000, E1   -29.991, E3 +490534.246}
SPL {X  -165.650, Y  +531.783, Z    +0.000, E1   -30.416, E3 +490544.139}
SPL {X  -165.650, Y  +534.115, Z    +0.000, E1   -30.089, E3 +490554.521}
SPL {X  -165.650, Y  +537.522, Z    +0.000, E1   -30.251, E3 +490565.436}
SPL {X  -165.650, Y  +540.621, Z    +0.000, E1   -30.014, E3 +490577.996}
SPL {X  -165.650, Y  +544.944, Z    +0.000, E1   -30.447, E3 +490590.196}
SPL {X  -165.650, Y  +547.199, Z    +0.000, E1   -30.132, E3 +490600.170}
SPL {X  -165.650, Y  +550.512, Z    +0.000, E1   -30.197, E3 +490611.495}
SPL {X  -165.650, Y  +553.852, Z    +0.000, E1   -30.156, E3 +490623.436}
SPL {X  -165.650, Y  +557.277, Z    +0.000, E1   -30.150, E3 +490635.611}
SPL {X  -165.650, Y  +561.168, Z    +0.000, E1   -30.194, E3 +490648.992}
SPL {X  -165.650, Y  +564.449, Z    +0.000, E1   -30.167, E3 +490660.675}
SPL {X  -165.650, Y  +566.935, Z    +0.000, E1   -30.135, E3 +490669.581}
SPL {X  -165.650, Y  +570.048, Z    +0.000, E1   -30.238, E3 +490679.906}
SPL {X  -165.650, Y  +573.110, Z    +0.000, E1   -30.057, E3 +490691.891}
SPL {X  -165.650, Y  +577.587, Z    +0.000, E1   -30.270, E3 +490706.330}
SPL {X  -165.650, Y  +581.190, Z    +0.000, E1   -30.107, E3 +490719.969}
SPL {X  -165.650, Y  +585.053, Z    +0.000, E1   -30.090, E3 +490733.839}
ENDSPLINE

SPLINE
SPL {X  -165.650, Y  +484.445, Z    +0.000, E1   +32.277, E3 +490751.244}
SPL {X  -165.650, Y  +481.524, Z    +0.000, E1   +31.089, E3 +490768.694}
SPL {X  -165.650, Y  +478.014, Z    +0.000, E1   +30.826, E3 +490782.302}
SPL {X  -165.650, Y  +474.473, Z    +0.000, E1   +30.943, E3 +490793.626}
SPL {X  -165.650, Y  +471.826, Z    +0.000, E1   +30.770, E3 +490803.810}
SPL {X  -165.650, Y  +467.753, Z    +0.000, E1   +30.878, E3 +490817.183}
SPL {X  -165.650, Y  +463.837, Z    +0.000, E1   +30.924, E3 +490830.117}
SPL {X  -165.650, Y  +461.106, Z    +0.000, E1   +30.916, E3 +490839.504}
SPL {X  -165.650, Y  +457.156, Z    +0.000, E1   +30.860, E3 +490853.581}
SPL {X  -165.650, Y  +453.156, Z    +0.000, E1   +30.934, E3 +490866.555}
SPL {X  -165.650, Y  +450.433, Z    +0.000, E1   +30.789, E3 +490876.910}
SPL {X  -165.650, Y  +447.097, Z    +0.000, E1   +30.843, E3 +490887.959}
SPL {X  -165.650, Y  +443.673, Z    +0.000, E1   +30.907, E3 +490899.266}
SPL {X  -165.650, Y  +439.486, Z    +0.000, E1   +30.857, E3 +490914.076}
SPL {X  -165.650, Y  +435.146, Z    +0.000, E1   +30.969, E3 +490927.995}
SPL {X  -165.650, Y  +431.607, Z    +0.000, E1   +30.889, E3 +490940.710}
SPL {X  -165.650, Y  +427.340, Z    +0.000, E1   +30.870, E3 +490955.421}
SPL {X  -165.650, Y  +423.901, Z    +0.000, E1   +30.858, E3 +490967.177}
SPL {X  -165.650, Y  +421.437, Z    +0.000, E1   +30.833, E3 +490975.776}
SPL {X  -165.650, Y  +418.489, Z    +0.000, E1   +30.835, E3 +490985.892}
SPL {X  -165.650, Y  +414.127, Z    +0.000, E1   +30.869, E3 +491000.801}
SPL {X  -165.650, Y  +408.547, Z    +0.000, E1   +30.964, E3 +491019.217}
SPL {X  -165.650, Y  +405.433, Z    +0.000, E1   +30.730, E3 +491031.194}
SPL {X  -165.650, Y  +401.473, Z    +0.000, E1   +30.933, E3 +491043.642}
SPL {X  -165.650, Y  +396.018, Z    +0.000, E1   +30.861, E3 +491062.827}
SPL {X  -165.650, Y  +391.522, Z    +0.000, E1   +30.837, E3 +491078.184}
SPL {X  -165.650, Y  +387.533, Z    +0.000, E1   +30.858, E3 +491091.810}
SPL {X  -165.650, Y  +383.627, Z    +0.000, E1   +30.885, E3 +491104.871}
SPL {X  -165.650, Y  +380.752, Z    +0.000, E1   +30.927, E3 +491114.384}
SPL {X  -165.648, Y  +377.739, Z    +0.000, E1   +30.835, E3 +491125.394}
SPL {X  -165.594, Y  +374.183, Z    +0.000, E1   +30.878, E3 +491137.231}
SPL {X  -165.429, Y  +369.945, Z    +0.000, E1   +30.850, E3 +491152.106}
SPL {X  -165.167, Y  +365.866, Z    +0.000, E1   +30.741, E3 +491166.638}
SPL {X  -164.892, Y  +362.671, Z    +0.000, E1   +30.830, E3 +491176.962}
SPL {X  -164.570, Y  +359.612, Z    +0.000, E1   +30.773, E3 +491187.775}
SPL {X  -164.104, Y  +355.923, Z    +0.000, E1   +30.626, E3 +491201.492}
SPL {X  -163.573, Y  +352.353, Z    +0.000, E1   +30.451, E3 +491214.756}
SPL {X  -162.976, Y  +348.856, Z    +0.000, E1   +30.757, E3 +491224.680}
SPL {X  -161.497, Y  +341.640, Z    +0.000, E1   +33.276, E3 +491231.958}
SPL {X  -152.976, Y  +314.952, Z    +0.000, E1   +38.607, E3 +491276.302}
SPL {X  -137.967, Y  +286.821, Z    +0.000, E1   +43.969, E3 +491319.523}
ENDSPLINE

SPLINE
SPL {X  -149.143, Y  +306.414, Z    +0.000, E1   +36.361, E3 +491370.656}
SPL {X  -164.268, Y  +357.145, Z    +0.000, E1   +15.880, E3 +491328.415}
SPL {X  -165.510, Y  +371.680, Z    +0.000, E1    +7.684, E3 +491331.417}
SPL {X  -165.628, Y  +375.818, Z    +0.000, E1    +5.016, E3 +491339.347}
SPL {X  -165.650, Y  +383.362, Z    +0.000, E1    +0.177, E3 +491320.380}
SPL {X  -165.650, Y  +383.923, Z    +0.000, E1    -0.215, E3 +491333.538}
SPL {X  -165.650, Y  +388.083, Z    +0.000, E1    -3.355, E3 +491332.401}
SPL {X  -165.650, Y  +395.510, Z    +0.000, E1    -9.810, E3 +491328.527}
SPL {X  -165.650, Y  +403.066, Z    +0.000, E1   -17.886, E3 +491321.361}
SPL {X  -165.650, Y  +416.345, Z    +0.000, E1   -29.511, E3 +491323.103}
SPL {X  -165.650, Y  +422.331, Z    +0.000, E1   -27.760, E3 +491348.602}
SPL {X  -165.650, Y  +441.276, Z    +0.000, E1   -37.343, E3 +491358.459}
SPL {X  -165.650, Y  +462.890, Z    +0.000, E1   -40.484, E3 +491392.542}
ENDSPLINE

SPLINE
SPL {X  -165.650, Y  +446.920, Z    +0.000, E1   -31.238, E3 +491404.868}
ENDSPLINE

SPLINE
SPL {X  -165.650, Y  +447.935, Z    +0.000, E1   -30.213, E3 +491415.156}
SPL {X  -165.650, Y  +451.020, Z    +0.000, E1   -30.224, E3 +491425.976}
SPL {X  -165.650, Y  +454.519, Z    +0.000, E1   -30.374, E3 +491437.159}
SPL {X  -165.650, Y  +457.429, Z    +0.000, E1   -30.029, E3 +491449.861}
SPL {X  -165.650, Y  +461.678, Z    +0.000, E1   -30.426, E3 +491461.985}
SPL {X  -165.650, Y  +463.853, Z    +0.000, E1   -30.103, E3 +491471.825}
SPL {X  -165.650, Y  +468.397, Z    +0.000, E1   -30.302, E3 +491486.629}
SPL {X  -165.650, Y  +472.566, Z    +0.000, E1   -30.124, E3 +491502.338}
SPL {X  -165.650, Y  +475.265, Z    +0.000, E1   -30.034, E3 +491512.375}
SPL {X  -165.650, Y  +477.862, Z    +0.000, E1   -30.319, E3 +491519.567}
SPL {X  -165.650, Y  +481.042, Z    +0.000, E1   -30.192, E3 +491531.827}
SPL {X  -165.650, Y  +485.236, Z    +0.000, E1   -30.294, E3 +491545.683}
SPL {X  -165.650, Y  +488.041, Z    +0.000, E1   -30.253, E3 +491555.804}
SPL {X  -165.650, Y  +491.281, Z    +0.000, E1   -30.148, E3 +491567.942}
SPL {X  -165.650, Y  +495.051, Z    +0.000, E1   -30.213, E3 +491580.751}
SPL {X  -165.650, Y  +499.546, Z    +0.000, E1   -30.283, E3 +491596.194}
SPL {X  -165.650, Y  +503.544, Z    +0.000, E1   -30.247, E3 +491610.262}
SPL {X  -165.650, Y  +506.344, Z    +0.000, E1   -30.129, E3 +491620.931}
SPL {X  -165.650, Y  +510.660, Z    +0.000, E1   -30.223, E3 +491635.634}
SPL {X  -165.650, Y  +514.670, Z    +0.000, E1   -30.278, E3 +491649.144}
SPL {X  -165.650, Y  +517.919, Z    +0.000, E1   -30.227, E3 +491661.004}
SPL {X  -165.650, Y  +522.822, Z    +0.000, E1   -30.289, E3 +491677.893}
SPL {X  -165.650, Y  +527.393, Z    +0.000, E1   -30.104, E3 +491695.141}
SPL {X  -165.650, Y  +531.783, Z    +0.000, E1   -30.416, E3 +491708.318}
SPL {X  -165.650, Y  +534.115, Z    +0.000, E1   -30.089, E3 +491718.700}
SPL {X  -165.650, Y  +537.522, Z    +0.000, E1   -30.251, E3 +491729.615}
SPL {X  -165.650, Y  +540.621, Z    +0.000, E1   -30.014, E3 +491742.176}
SPL {X  -165.650, Y  +544.944, Z    +0.000, E1   -30.447, E3 +491754.375}
SPL {X  -165.650, Y  +547.199, Z    +0.000, E1   -30.132, E3 +491764.349}
SPL {X  -165.650, Y  +550.512, Z    +0.000, E1   -30.197, E3 +491775.675}
SPL {X  -165.650, Y  +553.852, Z    +0.000, E1   -30.156, E3 +491787.615}
SPL {X  -165.650, Y  +557.277, Z    +0.000, E1   -30.150, E3 +491799.790}
SPL {X  -165.650, Y  +561.168, Z    +0.000, E1   -30.194, E3 +491813.171}
SPL {X  -165.650, Y  +565.528, Z    +0.000, E1   -30.192, E3 +491828.654}
SPL {X  -165.650, Y  +570.048, Z    +0.000, E1   -30.238, E3 +491844.085}
SPL {X  -165.650, Y  +573.110, Z    +0.000, E1   -30.057, E3 +491856.070}
SPL {X  -165.650, Y  +577.587, Z    +0.000, E1   -30.270, E3 +491870.509}
SPL {X  -165.650, Y  +581.190, Z    +0.000, E1   -30.107, E3 +491884.148}
SPL {X  -165.650, Y  +585.053, Z    +0.000, E1   -30.090, E3 +491898.019}
ENDSPLINE

SPLINE
SPL {X  -165.650, Y  +484.445, Z    +0.000, E1   +32.277, E3 +491915.423}
SPL {X  -165.650, Y  +481.524, Z    +0.000, E1   +31.089, E3 +491932.874}
SPL {X  -165.650, Y  +478.014, Z    +0.000, E1   +30.826, E3 +491946.481}
SPL {X  -165.650, Y  +474.473, Z    +0.000, E1   +30.943, E3 +491957.806}
SPL {X  -165.650, Y  +471.826, Z    +0.000, E1   +30.770, E3 +491967.989}
SPL {X  -165.650, Y  +467.753, Z    +0.000, E1   +30.878, E3 +491981.363}
SPL {X  -165.650, Y  +463.837, Z    +0.000, E1   +30.924, E3 +491994.296}
SPL {X  -165.650, Y  +461.106, Z    +0.000, E1   +30.916, E3 +492003.683}
SPL {X  -165.650, Y  +457.156, Z    +0.000, E1   +30.860, E3 +492017.760}
SPL {X  -165.650, Y  +453.156, Z    +0.000, E1   +30.934, E3 +492030.734}
SPL {X  -165.650, Y  +450.433, Z    +0.000, E1   +30.789, E3 +492041.089}
SPL {X  -165.650, Y  +447.097, Z    +0.000, E1   +30.843, E3 +492052.138}
SPL {X  -165.650, Y  +443.673, Z    +0.000, E1   +30.907, E3 +492063.445}
SPL {X  -165.650, Y  +439.486, Z    +0.000, E1   +30.857, E3 +492078.255}
SPL {X  -165.650, Y  +435.146, Z    +0.000, E1   +30.969, E3 +492092.174}
SPL {X  -165.650, Y  +431.607, Z    +0.000, E1   +30.889, E3 +492104.889}
SPL {X  -165.650, Y  +427.340, Z    +0.000, E1   +30.870, E3 +492119.600}
SPL {X  -165.650, Y  +423.901, Z    +0.000, E1   +30.858, E3 +492131.357}
SPL {X  -165.650, Y  +421.437, Z    +0.000, E1   +30.833, E3 +492139.955}
SPL {X  -165.650, Y  +418.489, Z    +0.000, E1   +30.835, E3 +492150.072}
SPL {X  -165.650, Y  +414.127, Z    +0.000, E1   +30.869, E3 +492164.980}
SPL {X  -165.650, Y  +408.547, Z    +0.000, E1   +30.964, E3 +492183.396}
SPL {X  -165.650, Y  +405.433, Z    +0.000, E1   +30.730, E3 +492195.373}
SPL {X  -165.650, Y  +401.473, Z    +0.000, E1   +30.933, E3 +492207.821}
SPL {X  -165.650, Y  +396.018, Z    +0.000, E1   +30.861, E3 +492227.006}
SPL {X  -165.650, Y  +390.331, Z    +0.000, E1   +30.892, E3 +492246.259}
SPL {X  -165.650, Y  +384.849, Z    +0.000, E1   +30.885, E3 +492265.062}
SPL {X  -165.650, Y  +380.752, Z    +0.000, E1   +30.927, E3 +492278.564}
SPL {X  -165.648, Y  +377.739, Z    +0.000, E1   +30.835, E3 +492289.573}
SPL {X  -165.594, Y  +374.183, Z    +0.000, E1   +30.878, E3 +492301.410}
SPL {X  -165.492, Y  +371.263, Z    +0.000, E1   +30.913, E3 +492311.105}
SPL {X  -165.379, Y  +369.027, Z    +0.000, E1   +30.727, E3 +492320.043}
SPL {X  -165.167, Y  +365.866, Z    +0.000, E1   +30.741, E3 +492330.817}
SPL {X  -164.892, Y  +362.671, Z    +0.000, E1   +30.830, E3 +492341.142}
SPL {X  -164.570, Y  +359.612, Z    +0.000, E1   +30.773, E3 +492351.954}
SPL {X  -164.104, Y  +355.923, Z    +0.000, E1   +30.626, E3 +492365.671}
SPL {X  -163.573, Y  +352.353, Z    +0.000, E1   +30.451, E3 +492378.935}
SPL {X  -162.476, Y  +346.230, Z    +0.000, E1   +31.677, E3 +492391.516}
SPL {X  -152.976, Y  +314.952, Z    +0.000, E1   +38.607, E3 +492440.481}
SPL {X  -137.967, Y  +286.821, Z    +0.000, E1   +43.969, E3 +492483.703}
ENDSPLINE

SPLINE
SPL {X  -153.316, Y  +315.777, Z    +0.000, E1   +33.140, E3 +492526.330}
SPL {X  -164.446, Y  +358.564, Z    +0.000, E1   +15.149, E3 +492491.541}
SPL {X  -165.379, Y  +369.025, Z    +0.000, E1    +9.158, E3 +492497.266}
SPL {X  -165.612, Y  +374.969, Z    +0.000, E1    +5.630, E3 +492499.941}
SPL {X  -165.650, Y  +383.362, Z    +0.000, E1    +0.177, E3 +492484.560}
SPL {X  -165.650, Y  +383.923, Z    +0.000, E1    -0.215, E3 +492497.717}
SPL {X  -165.650, Y  +388.083, Z    +0.000, E1    -3.355, E3 +492496.580}
SPL {X  -165.650, Y  +393.983, Z    +0.000, E1    -8.501, E3 +492492.979}
SPL {X  -165.650, Y  +402.241, Z    +0.000, E1   -16.711, E3 +492487.490}
SPL {X  -165.650, Y  +416.345, Z    +0.000, E1   -29.511, E3 +492487.282}
SPL {X  -165.650, Y  +422.331, Z    +0.000, E1   -27.760, E3 +492512.781}
SPL {X  -165.650, Y  +441.276, Z    +0.000, E1   -37.343, E3 +492522.639}
SPL {X  -165.650, Y  +462.890, Z    +0.000, E1   -40.484, E3 +492556.721}
ENDSPLINE

SPLINE
SPL {X  -165.650, Y  +446.920, Z    +0.000, E1   -31.238, E3 +492569.047}
ENDSPLINE

SPLINE
SPL {X  -165.650, Y  +447.935, Z    +0.000, E1   -30.213, E3 +492579.335}
SPL {X  -165.650, Y  +451.020, Z    +0.000, E1   -30.224, E3 +492590.156}
SPL {X  -165.650, Y  +454.519, Z    +0.000, E1   -30.374, E3 +492601.338}
SPL {X  -165.650, Y  +456.542, Z    +0.000, E1   -29.986, E3 +492611.083}
SPL {X  -165.650, Y  +460.618, Z    +0.000, E1   -30.298, E3 +492623.403}
SPL {X  -165.650, Y  +463.853, Z    +0.000, E1   -30.103, E3 +492636.004}
SPL {X  -165.650, Y  +467.246, Z    +0.000, E1   -30.279, E3 +492646.734}
SPL {X  -165.650, Y  +469.780, Z    +0.000, E1   -30.237, E3 +492655.859}
SPL {X  -165.650, Y  +472.566, Z    +0.000, E1   -30.124, E3 +492666.517}
SPL {X  -165.650, Y  +476.540, Z    +0.000, E1   -30.193, E3 +492680.061}
SPL {X  -165.650, Y  +480.320, Z    +0.000, E1   -30.163, E3 +492693.539}
SPL {X  -165.650, Y  +484.477, Z    +0.000, E1   -30.274, E3 +492707.428}
SPL {X  -165.650, Y  +488.041, Z    +0.000, E1   -30.253, E3 +492719.983}
SPL {X  -165.650, Y  +491.281, Z    +0.000, E1   -30.148, E3 +492732.122}
SPL {X  -165.650, Y  +495.051, Z    +0.000, E1   -30.213, E3 +492744.930}
SPL {X  -165.650, Y  +498.418, Z    +0.000, E1   -30.282, E3 +492756.223}
SPL {X  -165.650, Y  +500.833, Z    +0.000, E1   -30.191, E3 +492765.272}
SPL {X  -165.650, Y  +504.246, Z    +0.000, E1   -30.231, E3 +492777.138}
SPL {X  -165.650, Y  +507.017, Z    +0.000, E1   -30.108, E3 +492787.547}
SPL {X  -165.650, Y  +510.660, Z    +0.000, E1   -30.223, E3 +492799.813}
SPL {X  -165.650, Y  +515.918, Z    +0.000, E1   -30.316, E3 +492817.622}
SPL {X  -165.650, Y  +520.621, Z    +0.000, E1   -30.198, E3 +492834.907}
SPL {X  -165.650, Y  +525.344, Z    +0.000, E1   -30.269, E3 +492850.964}
SPL {X  -165.650, Y  +528.152, Z    +0.000, E1   -29.991, E3 +492862.605}
SPL {X  -165.650, Y  +531.783, Z    +0.000, E1   -30.416, E3 +492872.497}
SPL {X  -165.650, Y  +534.115, Z    +0.000, E1   -30.089, E3 +492882.879}
SPL {X  -165.650, Y  +538.363, Z    +0.000, E1   -30.232, E3 +492897.049}
SPL {X  -165.650, Y  +543.650, Z    +0.000, E1   -30.281, E3 +492915.269}
SPL {X  -165.650, Y  +547.199, Z    +0.000, E1   -30.132, E3 +492928.528}
SPL {X  -165.650, Y  +550.512, Z    +0.000, E1   -30.197, E3 +492939.854}
SPL {X  -165.650, Y  +554.908, Z    +0.000, E1   -30.180, E3 +492955.515}
SPL {X  -165.650, Y  +560.243, Z    +0.000, E1   -30.214, E3 +492974.141}
SPL {X  -165.650, Y  +565.528, Z    +0.000, E1   -30.192, E3 +492992.833}
SPL {X  -165.650, Y  +570.048, Z    +0.000, E1   -30.238, E3 +493008.264}
SPL {X  -165.650, Y  +573.110, Z    +0.000, E1   -30.057, E3 +493020.249}
SPL {X  -165.650, Y  +577.587, Z    +0.000, E1   -30.270, E3 +493034.688}
SPL {X  -165.650, Y  +581.190, Z    +0.000, E1   -30.107, E3 +493048.328}
SPL {X  -165.650, Y  +585.053, Z    +0.000, E1   -30.090, E3 +493062.198}
ENDSPLINE

SPLINE
SPL {X  -165.650, Y  +484.445, Z    +0.000, E1   +32.277, E3 +493079.602}
SPL {X  -165.650, Y  +481.524, Z    +0.000, E1   +31.089, E3 +493097.053}
SPL {X  -165.650, Y  +478.014, Z    +0.000, E1   +30.826, E3 +493110.660}
SPL {X  -165.650, Y  +474.473, Z    +0.000, E1   +30.943, E3 +493121.985}
SPL {X  -165.650, Y  +471.826, Z    +0.000, E1   +30.770, E3 +493132.168}
SPL {X  -165.650, Y  +467.753, Z    +0.000, E1   +30.878, E3 +493145.542}
SPL {X  -165.650, Y  +463.837, Z    +0.000, E1   +30.924, E3 +493158.475}
SPL {X  -165.650, Y  +461.106, Z    +0.000, E1   +30.916, E3 +493167.862}
SPL {X  -165.650, Y  +457.156, Z    +0.000, E1   +30.860, E3 +493181.939}
SPL {X  -165.650, Y  +453.156, Z    +0.000, E1   +30.934, E3 +493194.913}
SPL {X  -165.650, Y  +450.433, Z    +0.000, E1   +30.789, E3 +493205.268}
SPL {X  -165.650, Y  +447.097, Z    +0.000, E1   +30.843, E3 +493216.317}
SPL {X  -165.650, Y  +443.673, Z    +0.000, E1   +30.907, E3 +493227.624}
SPL {X  -165.650, Y  +439.486, Z    +0.000, E1   +30.857, E3 +493242.434}
SPL {X  -165.650, Y  +435.146, Z    +0.000, E1   +30.969, E3 +493256.353}
SPL {X  -165.650, Y  +431.607, Z    +0.000, E1   +30.889, E3 +493269.068}
SPL {X  -165.650, Y  +427.340, Z    +0.000, E1   +30.870, E3 +493283.779}
SPL {X  -165.650, Y  +423.901, Z    +0.000, E1   +30.858, E3 +493295.536}
SPL {X  -165.650, Y  +421.437, Z    +0.000, E1   +30.833, E3 +493304.134}
SPL {X  -165.650, Y  +418.489, Z    +0.000, E1   +30.835, E3 +493314.251}
SPL {X  -165.650, Y  +414.127, Z    +0.000, E1   +30.869, E3 +493329.159}
SPL {X  -165.650, Y  +408.547, Z    +0.000, E1   +30.964, E3 +493347.575}
SPL {X  -165.650, Y  +405.433, Z    +0.000, E1   +30.730, E3 +493359.552}
SPL {X  -165.650, Y  +401.473, Z    +0.000, E1   +30.933, E3 +493372.001}
SPL {X  -165.650, Y  +396.018, Z    +0.000, E1   +30.861, E3 +493391.185}
SPL {X  -165.650, Y  +390.331, Z    +0.000, E1   +30.892, E3 +493410.438}
SPL {X  -165.650, Y  +384.849, Z    +0.000, E1   +30.885, E3 +493429.241}
SPL {X  -165.650, Y  +380.752, Z    +0.000, E1   +30.927, E3 +493442.743}
SPL {X  -165.648, Y  +377.739, Z    +0.000, E1   +30.835, E3 +493453.752}
SPL {X  -165.594, Y  +374.183, Z    +0.000, E1   +30.878, E3 +493465.589}
SPL {X  -165.492, Y  +371.263, Z    +0.000, E1   +30.913, E3 +493475.284}
SPL {X  -165.379, Y  +369.027, Z    +0.000, E1   +30.727, E3 +493484.223}
SPL {X  -165.167, Y  +365.866, Z    +0.000, E1   +30.741, E3 +493494.997}
SPL {X  -164.892, Y  +362.671, Z    +0.000, E1   +30.830, E3 +493505.321}
SPL {X  -164.570, Y  +359.612, Z    +0.000, E1   +30.773, E3 +493516.133}
SPL {X  -164.104, Y  +355.923, Z    +0.000, E1   +30.626, E3 +493529.850}
SPL {X  -163.573, Y  +352.353, Z    +0.000, E1   +30.451, E3 +493543.115}
SPL {X  -162.476, Y  +346.230, Z    +0.000, E1   +31.677, E3 +493555.695}
SPL {X  -152.976, Y  +314.952, Z    +0.000, E1   +38.607, E3 +493604.661}
SPL {X  -137.967, Y  +286.821, Z    +0.000, E1   +43.969, E3 +493647.882}
ENDSPLINE

SPLINE
SPL {X  -153.316, Y  +315.777, Z    +0.000, E1   +33.140, E3 +493690.509}
SPL {X  -164.446, Y  +358.564, Z    +0.000, E1   +15.149, E3 +493655.720}
SPL {X  -165.510, Y  +371.680, Z    +0.000, E1    +7.684, E3 +493659.776}
SPL {X  -165.628, Y  +375.818, Z    +0.000, E1    +5.016, E3 +493667.705}
SPL {X  -165.650, Y  +383.362, Z    +0.000, E1    +0.177, E3 +493648.739}
SPL {X  -165.650, Y  +383.923, Z    +0.000, E1    -0.215, E3 +493661.896}
SPL {X  -165.650, Y  +388.083, Z    +0.000, E1    -3.355, E3 +493660.760}
SPL {X  -165.650, Y  +393.983, Z    +0.000, E1    -8.501, E3 +493657.158}
SPL {X  -165.650, Y  +402.241, Z    +0.000, E1   -16.711, E3 +493651.670}
SPL {X  -165.650, Y  +416.345, Z    +0.000, E1   -29.511, E3 +493651.462}
SPL {X  -165.650, Y  +422.331, Z    +0.000, E1   -27.760, E3 +493676.961}
SPL {X  -165.650, Y  +441.276, Z    +0.000, E1   -37.343, E3 +493686.818}
SPL {X  -165.650, Y  +462.890, Z    +0.000, E1   -40.484, E3 +493720.901}
ENDSPLINE

SPLINE
SPL {X  -165.650, Y  +446.920, Z    +0.000, E1   -31.238, E3 +493733.226}
ENDSPLINE

SPLINE
SPL {X  -165.650, Y  +447.935, Z    +0.000, E1   -30.213, E3 +493743.514}
SPL {X  -165.650, Y  +451.020, Z    +0.000, E1   -30.224, E3 +493754.335}
SPL {X  -165.650, Y  +454.519, Z    +0.000, E1   -30.374, E3 +493765.517}
SPL {X  -165.650, Y  +456.542, Z    +0.000, E1   -29.986, E3 +493775.262}
SPL {X  -165.650, Y  +460.618, Z    +0.000, E1   -30.298, E3 +493787.582}
SPL {X  -165.650, Y  +463.853, Z    +0.000, E1   -30.103, E3 +493800.183}
SPL {X  -165.650, Y  +468.397, Z    +0.000, E1   -30.302, E3 +493814.987}
SPL {X  -165.650, Y  +472.566, Z    +0.000, E1   -30.124, E3 +493830.696}
SPL {X  -165.650, Y  +475.265, Z    +0.000, E1   -30.034, E3 +493840.734}
SPL {X  -165.650, Y  +477.862, Z    +0.000, E1   -30.319, E3 +493847.925}
SPL {X  -165.650, Y  +481.042, Z    +0.000, E1   -30.192, E3 +493860.186}
SPL {X  -165.650, Y  +485.236, Z    +0.000, E1   -30.294, E3 +493874.041}
SPL {X  -165.650, Y  +488.041, Z    +0.000, E1   -30.253, E3 +493884.162}
SPL {X  -165.650, Y  +491.281, Z    +0.000, E1   -30.148, E3 +493896.301}
SPL {X  -165.650, Y  +495.051, Z    +0.000, E1   -30.213, E3 +493909.109}
SPL {X  -165.650, Y  +499.546, Z    +0.000, E1   -30.283, E3 +493924.552}
SPL {X  -165.650, Y  +503.544, Z    +0.000, E1   -30.247, E3 +493938.620}
SPL {X  -165.650, Y  +506.344, Z    +0.000, E1   -30.129, E3 +493949.289}
SPL {X  -165.650, Y  +510.660, Z    +0.000, E1   -30.223, E3 +493963.993}
SPL {X  -165.650, Y  +514.670, Z    +0.000, E1   -30.278, E3 +493977.502}
SPL {X  -165.650, Y  +517.919, Z    +0.000, E1   -30.227, E3 +493989.362}
SPL {X  -165.650, Y  +521.521, Z    +0.000, E1   -30.210, E3 +494002.036}
SPL {X  -165.650, Y  +525.344, Z    +0.000, E1   -30.269, E3 +494015.143}
SPL {X  -165.650, Y  +528.152, Z    +0.000, E1   -29.991, E3 +494026.784}
SPL {X  -165.650, Y  +531.783, Z    +0.000, E1   -30.416, E3 +494036.676}
SPL {X  -165.650, Y  +534.115, Z    +0.000, E1   -30.089, E3 +494047.059}
SPL {X  -165.650, Y  +537.522, Z    +0.000, E1   -30.251, E3 +494057.973}
SPL {X  -165.650, Y  +540.621, Z    +0.000, E1   -30.014, E3 +494070.534}
SPL {X  -165.650, Y  +544.944, Z    +0.000, E1   -30.447, E3 +494082.733}
SPL {X  -165.650, Y  +548.549, Z    +0.000, E1   -30.216, E3 +494097.057}
SPL {X  -165.650, Y  +553.092, Z    +0.000, E1   -30.157, E3 +494113.399}
SPL {X  -165.650, Y  +557.277, Z    +0.000, E1   -30.150, E3 +494128.148}
SPL {X  -165.650, Y  +561.168, Z    +0.000, E1   -30.194, E3 +494141.529}
SPL {X  -165.650, Y  +564.449, Z    +0.000, E1   -30.167, E3 +494153.213}
SPL {X  -165.650, Y  +566.935, Z    +0.000, E1   -30.135, E3 +494162.118}
SPL {X  -165.650, Y  +570.048, Z    +0.000, E1   -30.238, E3 +494172.443}
SPL {X  -165.650, Y  +573.110, Z    +0.000, E1   -30.057, E3 +494184.428}
SPL {X  -165.650, Y  +576.497, Z    +0.000, E1   -30.234, E3 +494195.126}
SPL {X  -165.650, Y  +580.354, Z    +0.000, E1   -30.196, E3 +494209.141}
SPL {X  -165.650, Y  +585.053, Z    +0.000, E1   -30.090, E3 +494226.377}
ENDSPLINE

SPLINE
SPL {X  -165.650, Y  +484.445, Z    +0.000, E1   +32.277, E3 +494243.781}
SPL {X  -165.650, Y  +481.524, Z    +0.000, E1   +31.089, E3 +494261.232}
SPL {X  -165.650, Y  +478.014, Z    +0.000, E1   +30.826, E3 +494274.839}
SPL {X  -165.650, Y  +474.473, Z    +0.000, E1   +30.943, E3 +494286.164}
SPL {X  -165.650, Y  +470.376, Z    +0.000, E1   +30.888, E3 +494300.693}
SPL {X  -165.650, Y  +465.146, Z    +0.000, E1   +30.883, E3 +494318.624}
SPL {X  -165.650, Y  +461.106, Z    +0.000, E1   +30.916, E3 +494332.042}
SPL {X  -165.650, Y  +458.435, Z    +0.000, E1   +30.759, E3 +494342.250}
SPL {X  -165.650, Y  +454.220, Z    +0.000, E1   +30.954, E3 +494355.483}
SPL {X  -165.650, Y  +450.433, Z    +0.000, E1   +30.789, E3 +494369.447}
SPL {X  -165.650, Y  +447.097, Z    +0.000, E1   +30.843, E3 +494380.496}
SPL {X  -165.650, Y  +443.673, Z    +0.000, E1   +30.907, E3 +494391.804}
SPL {X  -165.650, Y  +440.976, Z    +0.000, E1   +30.719, E3 +494402.260}
SPL {X  -165.650, Y  +437.973, Z    +0.000, E1   +30.928, E3 +494411.133}
SPL {X  -165.650, Y  +434.043, Z    +0.000, E1   +30.950, E3 +494424.629}
SPL {X  -165.650, Y  +430.419, Z    +0.000, E1   +30.895, E3 +494437.132}
SPL {X  -165.650, Y  +427.340, Z    +0.000, E1   +30.870, E3 +494447.959}
SPL {X  -165.650, Y  +422.641, Z    +0.000, E1   +30.884, E3 +494464.048}
SPL {X  -165.650, Y  +418.489, Z    +0.000, E1   +30.835, E3 +494478.430}
SPL {X  -165.650, Y  +414.127, Z    +0.000, E1   +30.869, E3 +494493.338}
SPL {X  -165.650, Y  +408.547, Z    +0.000, E1   +30.964, E3 +494511.754}
SPL {X  -165.650, Y  +405.433, Z    +0.000, E1   +30.730, E3 +494523.731}
SPL {X  -165.650, Y  +402.516, Z    +0.000, E1   +30.874, E3 +494532.854}
SPL {X  -165.650, Y  +398.147, Z    +0.000, E1   +30.902, E3 +494547.732}
SPL {X  -165.650, Y  +394.694, Z    +0.000, E1   +30.805, E3 +494560.041}
SPL {X  -165.650, Y  +391.522, Z    +0.000, E1   +30.837, E3 +494570.721}
SPL {X  -165.650, Y  +387.533, Z    +0.000, E1   +30.858, E3 +494584.348}
SPL {X  -165.650, Y  +383.627, Z    +0.000, E1   +30.885, E3 +494597.408}
SPL {X  -165.650, Y  +379.886, Z    +0.000, E1   +30.887, E3 +494610.296}
SPL {X  -165.614, Y  +375.058, Z    +0.000, E1   +30.905, E3 +494626.749}
SPL {X  -165.492, Y  +371.263, Z    +0.000, E1   +30.913, E3 +494639.463}
SPL {X  -165.379, Y  +369.027, Z    +0.000, E1   +30.727, E3 +494648.402}
SPL {X  -165.167, Y  +365.866, Z    +0.000, E1   +30.741, E3 +494659.176}
SPL {X  -164.892, Y  +362.671, Z    +0.000, E1   +30.830, E3 +494669.500}
SPL {X  -164.570, Y  +359.612, Z    +0.000, E1   +30.773, E3 +494680.312}
SPL {X  -164.104, Y  +355.923, Z    +0.000, E1   +30.626, E3 +494694.029}
SPL {X  -163.573, Y  +352.353, Z    +0.000, E1   +30.451, E3 +494707.294}
SPL {X  -162.976, Y  +348.856, Z    +0.000, E1   +30.757, E3 +494717.217}
SPL {X  -161.497, Y  +341.640, Z    +0.000, E1   +33.276, E3 +494724.495}
SPL {X  -152.976, Y  +314.952, Z    +0.000, E1   +38.607, E3 +494768.840}
SPL {X  -137.967, Y  +286.821, Z    +0.000, E1   +43.969, E3 +494812.061}
ENDSPLINE

SPLINE
SPL {X  -149.143, Y  +306.414, Z    +0.000, E1   +36.361, E3 +494863.193}
SPL {X  -164.268, Y  +357.145, Z    +0.000, E1   +15.880, E3 +494820.952}
SPL {X  -165.379, Y  +369.025, Z    +0.000, E1    +9.158, E3 +494825.624}
SPL {X  -165.612, Y  +374.969, Z    +0.000, E1    +5.630, E3 +494828.299}
SPL {X  -165.650, Y  +383.362, Z    +0.000, E1    +0.177, E3 +494812.918}
SPL {X  -165.650, Y  +383.923, Z    +0.000, E1    -0.215, E3 +494826.075}
SPL {X  -165.650, Y  +388.083, Z    +0.000, E1    -3.355, E3 +494824.939}
SPL {X  -165.650, Y  +393.983, Z    +0.000, E1    -8.501, E3 +494821.337}
SPL {X  -165.650, Y  +402.241, Z    +0.000, E1   -16.711, E3 +494815.849}
SPL {X  -165.650, Y  +416.345, Z    +0.000, E1   -29.511, E3 +494815.641}
SPL {X  -165.650, Y  +422.331, Z    +0.000, E1   -27.760, E3 +494841.140}
SPL {X  -165.650, Y  +441.276, Z    +0.000, E1   -37.343, E3 +494850.997}
SPL {X  -165.650, Y  +462.890, Z    +0.000, E1   -40.484, E3 +494885.080}
ENDSPLINE

SPLINE
SPL {X  -165.650, Y  +446.920, Z    +0.000, E1   -31.238, E3 +494897.405}
ENDSPLINE

SPLINE
SPL {X  -165.650, Y  +447.935, Z    +0.000, E1   -30.213, E3 +494907.693}
SPL {X  -165.650, Y  +451.020, Z    +0.000, E1   -30.224, E3 +494918.514}
SPL {X  -165.650, Y  +454.519, Z    +0.000, E1   -30.374, E3 +494929.696}
SPL {X  -165.650, Y  +456.542, Z    +0.000, E1   -29.986, E3 +494939.441}
SPL {X  -165.650, Y  +460.618, Z    +0.000, E1   -30.298, E3 +494951.761}
SPL {X  -165.650, Y  +463.853, Z    +0.000, E1   -30.103, E3 +494964.362}
SPL {X  -165.650, Y  +467.246, Z    +0.000, E1   -30.279, E3 +494975.092}
SPL {X  -165.650, Y  +469.780, Z    +0.000, E1   -30.237, E3 +494984.218}
SPL {X  -165.650, Y  +472.566, Z    +0.000, E1   -30.124, E3 +494994.875}
SPL {X  -165.650, Y  +476.540, Z    +0.000, E1   -30.193, E3 +495008.419}
SPL {X  -165.650, Y  +480.320, Z    +0.000, E1   -30.163, E3 +495021.897}
SPL {X  -165.650, Y  +484.477, Z    +0.000, E1   -30.274, E3 +495035.786}
SPL {X  -165.650, Y  +488.041, Z    +0.000, E1   -30.253, E3 +495048.342}
SPL {X  -165.650, Y  +491.281, Z    +0.000, E1   -30.148, E3 +495060.480}
SPL {X  -165.650, Y  +495.051, Z    +0.000, E1   -30.213, E3 +495073.288}
SPL {X  -165.650, Y  +498.418, Z    +0.000, E1   -30.282, E3 +495084.581}
SPL {X  -165.650, Y  +502.421, Z    +0.000, E1   -30.263, E3 +495098.939}
SPL {X  -165.650, Y  +506.344, Z    +0.000, E1   -30.129, E3 +495113.468}
SPL {X  -165.650, Y  +509.866, Z    +0.000, E1   -30.236, E3 +495125.137}
SPL {X  -165.650, Y  +513.685, Z    +0.000, E1   -30.234, E3 +495138.634}
SPL {X  -165.650, Y  +517.104, Z    +0.000, E1   -30.280, E3 +495150.185}
SPL {X  -165.650, Y  +520.621, Z    +0.000, E1   -30.198, E3 +495163.265}
SPL {X  -165.650, Y  +525.344, Z    +0.000, E1   -30.269, E3 +495179.322}
SPL {X  -165.650, Y  +528.152, Z    +0.000, E1   -29.991, E3 +495190.963}
SPL {X  -165.650, Y  +531.783, Z    +0.000, E1   -30.416, E3 +495200.856}
SPL {X  -165.650, Y  +534.115, Z    +0.000, E1   -30.089, E3 +495211.238}
SPL {X  -165.650, Y  +537.522, Z    +0.000, E1   -30.251, E3 +495222.152}
SPL {X  -165.650, Y  +540.621, Z    +0.000, E1   -30.014, E3 +495234.713}
SPL {X  -165.650, Y  +544.944, Z    +0.000, E1   -30.447, E3 +495246.913}
SPL {X  -165.650, Y  +548.549, Z    +0.000, E1   -30.216, E3 +495261.236}
SPL {X  -165.650, Y  +553.092, Z    +0.000, E1   -30.157, E3 +495277.578}
SPL {X  -165.650, Y  +557.277, Z    +0.000, E1   -30.150, E3 +495292.327}
SPL {X  -165.650, Y  +561.168, Z    +0.000, E1   -30.194, E3 +495305.709}
SPL {X  -165.650, Y  +564.449, Z    +0.000, E1   -30.167, E3 +495317.392}
SPL {X  -165.650, Y  +566.935, Z    +0.000, E1   -30.135, E3 +495326.297}
SPL {X  -165.650, Y  +570.048, Z    +0.000, E1   -30.238, E3 +495336.622}
SPL {X  -165.650, Y  +573.110, Z    +0.000, E1   -30.057, E3 +495348.607}
SPL {X  -165.650, Y  +577.587, Z    +0.000, E1   -30.270, E3 +495363.046}
SPL {X  -165.650, Y  +581.190, Z    +0.000, E1   -30.107, E3 +495376.686}
SPL {X  -165.650, Y  +585.053, Z    +0.000, E1   -30.090, E3 +495390.556}
ENDSPLINE

SPLINE
SPL {X  -165.650, Y  +484.968, Z    +0.000, E1   +32.508, E3 +495404.522}
SPL {X  -165.650, Y  +482.515, Z    +0.000, E1   +31.539, E3 +495419.050}
SPL {X  -165.650, Y  +479.127, Z    +0.000, E1   +30.804, E3 +495435.514}
SPL {X  -165.650, Y  +474.473, Z    +0.000, E1   +30.943, E3 +495450.343}
SPL {X  -165.650, Y  +470.376, Z    +0.000, E1   +30.888, E3 +495464.872}
SPL {X  -165.650, Y  +465.146, Z    +0.000, E1   +30.883, E3 +495482.803}
SPL {X  -165.650, Y  +461.106, Z    +0.000, E1   +30.916, E3 +495496.221}
SPL {X  -165.650, Y  +457.156, Z    +0.000, E1   +30.860, E3 +495510.297}
SPL {X  -165.650, Y  +453.156, Z    +0.000, E1   +30.934, E3 +495523.271}
SPL {X  -165.650, Y  +450.433, Z    +0.000, E1   +30.789, E3 +495533.627}
SPL {X  -165.650, Y  +447.097, Z    +0.000, E1   +30.843, E3 +495544.675}
SPL {X  -165.650, Y  +443.673, Z    +0.000, E1   +30.907, E3 +495555.983}
SPL {X  -165.650, Y  +439.486, Z    +0.000, E1   +30.857, E3 +495570.792}
SPL {X  -165.650, Y  +435.146, Z    +0.000, E1   +30.969, E3 +495584.711}
SPL {X  -165.650, Y  +431.607, Z    +0.000, E1   +30.889, E3 +495597.426}
SPL {X  -165.650, Y  +427.340, Z    +0.000, E1   +30.870, E3 +495612.138}
SPL {X  -165.650, Y  +423.901, Z    +0.000, E1   +30.858, E3 +495623.894}
SPL {X  -165.650, Y  +421.437, Z    +0.000, E1   +30.833, E3 +495632.492}
SPL {X  -165.650, Y  +418.489, Z    +0.000, E1   +30.835, E3 +495642.609}
SPL {X  -165.650, Y  +414.127, Z    +0.000, E1   +30.869, E3 +495657.517}
SPL {X  -165.650, Y  +408.547, Z    +0.000, E1   +30.964, E3 +495675.933}
SPL {X  -165.650, Y  +405.433, Z    +0.000, E1   +30.730, E3 +495687.910}
SPL {X  -165.650, Y  +402.516, Z    +0.000, E1   +30.874, E3 +495697.033}
SPL {X  -165.650, Y  +398.147, Z    +0.000, E1   +30.902, E3 +495711.911}
SPL {X  -165.650, Y  +394.694, Z    +0.000, E1   +30.805, E3 +495724.220}
SPL {X  -165.650, Y  +391.522, Z    +0.000, E1   +30.837, E3 +495734.901}
SPL {X  -165.650, Y  +387.533, Z    +0.000, E1   +30.858, E3 +495748.527}
SPL {X  -165.650, Y  +383.627, Z    +0.000, E1   +30.885, E3 +495761.587}
SPL {X  -165.650, Y  +379.886, Z    +0.000, E1   +30.887, E3 +495774.475}
SPL {X  -165.614, Y  +375.058, Z    +0.000, E1   +30.905, E3 +495790.928}
SPL {X  -165.492, Y  +371.263, Z    +0.000, E1   +30.913, E3 +495803.642}
SPL {X  -165.379, Y  +369.027, Z    +0.000, E1   +30.727, E3 +495812.581}
SPL {X  -165.167, Y  +365.866, Z    +0.000, E1   +30.741, E3 +495823.355}
SPL {X  -164.892, Y  +362.671, Z    +0.000, E1   +30.830, E3 +495833.679}
SPL {X  -164.570, Y  +359.612, Z    +0.000, E1   +30.773, E3 +495844.492}
SPL {X  -164.104, Y  +355.923, Z    +0.000, E1   +30.626, E3 +495858.208}
SPL {X  -163.573, Y  +352.353, Z    +0.000, E1   +30.451, E3 +495871.473}
SPL {X  -162.476, Y  +346.230, Z    +0.000, E1   +31.677, E3 +495884.054}
SPL {X  -152.976, Y  +314.952, Z    +0.000, E1   +38.607, E3 +495933.019}
SPL {X  -137.967, Y  +286.821, Z    +0.000, E1   +43.969, E3 +495976.240}
ENDSPLINE

SPLINE
SPL {X  -153.316, Y  +315.777, Z    +0.000, E1   +33.140, E3 +496018.867}
SPL {X  -164.446, Y  +358.564, Z    +0.000, E1   +15.149, E3 +495984.078}
SPL {X  -165.510, Y  +371.680, Z    +0.000, E1    +7.684, E3 +495988.134}
SPL {X  -165.628, Y  +375.818, Z    +0.000, E1    +5.016, E3 +495996.063}
SPL {X  -165.650, Y  +383.362, Z    +0.000, E1    +0.177, E3 +495977.097}
SPL {X  -165.650, Y  +383.923, Z    +0.000, E1    -0.215, E3 +495990.254}
SPL {X  -165.650, Y  +388.083, Z    +0.000, E1    -3.355, E3 +495989.118}
SPL {X  -165.650, Y  +393.983, Z    +0.000, E1    -8.501, E3 +495985.516}
SPL {X  -165.650, Y  +402.241, Z    +0.000, E1   -16.711, E3 +495980.028}
SPL {X  -165.650, Y  +416.345, Z    +0.000, E1   -29.511, E3 +495979.820}
SPL {X  -165.650, Y  +422.331, Z    +0.000, E1   -27.760, E3 +496005.319}
SPL {X  -165.650, Y  +435.050, Z    +0.000, E1   -34.610, E3 +496011.821}
SPL {X  -165.650, Y  +446.725, Z    +0.000, E1   -39.593, E3 +496018.083}
SPL {X  -165.650, Y  +462.890, Z    +0.000, E1   -40.484, E3 +496049.259}
ENDSPLINE

SPLINE
SPL {X  -165.650, Y  +446.920, Z    +0.000, E1   -31.238, E3 +496061.585}
ENDSPLINE

SPLINE
SPL {X  -165.650, Y  +447.935, Z    +0.000, E1   -30.213, E3 +496071.873}
SPL {X  -165.650, Y  +451.020, Z    +0.000, E1   -30.224, E3 +496082.693}
SPL {X  -165.650, Y  +454.519, Z    +0.000, E1   -30.374, E3 +496093.875}
SPL {X  -165.650, Y  +456.542, Z    +0.000, E1   -29.986, E3 +496103.620}
SPL {X  -165.650, Y  +460.618, Z    +0.000, E1   -30.298, E3 +496115.940}
SPL {X  -165.650, Y  +463.853, Z    +0.000, E1   -30.103, E3 +496128.541}
SPL {X  -165.650, Y  +467.246, Z    +0.000, E1   -30.279, E3 +496139.271}
SPL {X  -165.650, Y  +469.780, Z    +0.000, E1   -30.237, E3 +496148.397}
SPL {X  -165.650, Y  +472.566, Z    +0.000, E1   -30.124, E3 +496159.054}
SPL {X  -165.650, Y  +476.540, Z    +0.000, E1   -30.193, E3 +496172.598}
SPL {X  -165.650, Y  +480.320, Z    +0.000, E1   -30.163, E3 +496186.076}
SPL {X  -165.650, Y  +484.477, Z    +0.000, E1   -30.274, E3 +496199.966}
SPL {X  -165.650, Y  +489.057, Z    +0.000, E1   -30.341, E3 +496215.605}
SPL {X  -165.650, Y  +491.647, Z    +0.000, E1   -29.894, E3 +496227.538}
SPL {X  -165.650, Y  +495.051, Z    +0.000, E1   -30.213, E3 +496237.467}
SPL {X  -165.650, Y  +499.546, Z    +0.000, E1   -30.283, E3 +496252.910}
SPL {X  -165.650, Y  +503.544, Z    +0.000, E1   -30.247, E3 +496266.979}
SPL {X  -165.650, Y  +506.344, Z    +0.000, E1   -30.129, E3 +496277.647}
SPL {X  -165.650, Y  +510.660, Z    +0.000, E1   -30.223, E3 +496292.351}
SPL {X  -165.650, Y  +514.670, Z    +0.000, E1   -30.278, E3 +496305.860}
SPL {X  -165.650, Y  +517.919, Z    +0.000, E1   -30.227, E3 +496317.720}
SPL {X  -165.650, Y  +521.521, Z    +0.000, E1   -30.210, E3 +496330.395}
SPL {X  -165.650, Y  +525.344, Z    +0.000, E1   -30.269, E3 +496343.501}
SPL {X  -165.650, Y  +528.152, Z    +0.000, E1   -29.991, E3 +496355.142}
SPL {X  -165.650, Y  +531.783, Z    +0.000, E1   -30.416, E3 +496365.035}
SPL {X  -165.650, Y  +534.115, Z    +0.000, E1   -30.089, E3 +496375.417}
SPL {X  -165.650, Y  +537.522, Z    +0.000, E1   -30.251, E3 +496386.331}
SPL {X  -165.650, Y  +540.621, Z    +0.000, E1   -30.014, E3 +496398.892}
SPL {X  -165.650, Y  +544.944, Z    +0.000, E1   -30.447, E3 +496411.092}
SPL {X  -165.650, Y  +547.199, Z    +0.000, E1   -30.132, E3 +496421.065}
SPL {X  -165.650, Y  +550.512, Z    +0.000, E1   -30.197, E3 +496432.391}
SPL {X  -165.650, Y  +553.852, Z    +0.000, E1   -30.156, E3 +496444.332}
SPL {X  -165.650, Y  +557.277, Z    +0.000, E1   -30.150, E3 +496456.506}
SPL {X  -165.650, Y  +561.168, Z    +0.000, E1   -30.194, E3 +496469.888}
SPL {X  -165.650, Y  +565.528, Z    +0.000, E1   -30.192, E3 +496485.370}
SPL {X  -165.650, Y  +570.048, Z    +0.000, E1   -30.238, E3 +496500.802}
SPL {X  -165.650, Y  +573.110, Z    +0.000, E1   -30.057, E3 +496512.786}
SPL {X  -165.650, Y  +577.587, Z    +0.000, E1   -30.270, E3 +496527.225}
SPL {X  -165.650, Y  +581.190, Z    +0.000, E1   -30.107, E3 +496540.865}
SPL {X  -165.650, Y  +585.053, Z    +0.000, E1   -30.090, E3 +496554.735}
ENDSPLINE

SPLINE
SPL {X  -165.650, Y  +484.445, Z    +0.000, E1   +32.277, E3 +496572.139}
SPL {X  -165.650, Y  +481.524, Z    +0.000, E1   +31.089, E3 +496589.590}
SPL {X  -165.650, Y  +478.014, Z    +0.000, E1   +30.826, E3 +496603.198}
SPL {X  -165.650, Y  +474.473, Z    +0.000, E1   +30.943, E3 +496614.522}
SPL {X  -165.650, Y  +471.826, Z    +0.000, E1   +30.770, E3 +496624.706}
SPL {X  -165.650, Y  +467.753, Z    +0.000, E1   +30.878, E3 +496638.079}
SPL {X  -165.650, Y  +463.837, Z    +0.000, E1   +30.924, E3 +496651.013}
SPL {X  -165.650, Y  +461.106, Z    +0.000, E1   +30.916, E3 +496660.400}
SPL {X  -165.650, Y  +457.156, Z    +0.000, E1   +30.860, E3 +496674.476}
SPL {X  -165.650, Y  +453.156, Z    +0.000, E1   +30.934, E3 +496687.450}
SPL {X  -165.650, Y  +450.433, Z    +0.000, E1   +30.789, E3 +496697.806}
SPL {X  -165.650, Y  +447.097, Z    +0.000, E1   +30.843, E3 +496708.854}
SPL {X  -165.650, Y  +443.673, Z    +0.000, E1   +30.907, E3 +496720.162}
SPL {X  -165.650, Y  +439.486, Z    +0.000, E1   +30.857, E3 +496734.971}
SPL {X  -165.650, Y  +435.146, Z    +0.000, E1   +30.969, E3 +496748.890}
SPL {X  -165.650, Y  +431.607, Z    +0.000, E1   +30.889, E3 +496761.605}
SPL {X  -165.650, Y  +427.340, Z    +0.000, E1   +30.870, E3 +496776.317}
SPL {X  -165.650, Y  +423.901, Z    +0.000, E1   +30.858, E3 +496788.073}
SPL {X  -165.650, Y  +421.437, Z    +0.000, E1   +30.833, E3 +496796.671}
SPL {X  -165.650, Y  +418.489, Z    +0.000, E1   +30.835, E3 +496806.788}
SPL {X  -165.650, Y  +414.127, Z    +0.000, E1   +30.869, E3 +496821.697}
SPL {X  -165.650, Y  +408.547, Z    +0.000, E1   +30.964, E3 +496840.112}
SPL {X  -165.650, Y  +405.433, Z    +0.000, E1   +30.730, E3 +496852.089}
SPL {X  -165.650, Y  +401.473, Z    +0.000, E1   +30.933, E3 +496864.538}
SPL {X  -165.650, Y  +396.018, Z    +0.000, E1   +30.861, E3 +496883.723}
SPL {X  -165.650, Y  +391.522, Z    +0.000, E1   +30.837, E3 +496899.080}
SPL {X  -165.650, Y  +387.533, Z    +0.000, E1   +30.858, E3 +496912.706}
SPL {X  -165.650, Y  +383.627, Z    +0.000, E1   +30.885, E3 +496925.766}
SPL {X  -165.650, Y  +380.752, Z    +0.000, E1   +30.927, E3 +496935.280}
SPL {X  -165.648, Y  +377.739, Z    +0.000, E1   +30.835, E3 +496946.290}
SPL {X  -165.594, Y  +374.183, Z    +0.000, E1   +30.878, E3 +496958.126}
SPL {X  -165.429, Y  +369.945, Z    +0.000, E1   +30.850, E3 +496973.001}
SPL {X  -165.167, Y  +365.866, Z    +0.000, E1   +30.741, E3 +496987.534}
SPL {X  -164.892, Y  +362.671, Z    +0.000, E1   +30.830, E3 +496997.858}
SPL {X  -164.570, Y  +359.612, Z    +0.000, E1   +30.773, E3 +497008.671}
SPL {X  -164.104, Y  +355.923, Z    +0.000, E1   +30.626, E3 +497022.387}
SPL {X  -163.573, Y  +352.353, Z    +0.000, E1   +30.451, E3 +497035.652}
SPL {X  -162.976, Y  +348.856, Z    +0.000, E1   +30.757, E3 +497045.576}
SPL {X  -161.497, Y  +341.640, Z    +0.000, E1   +33.276, E3 +497052.853}
SPL {X  -152.976, Y  +314.952, Z    +0.000, E1   +38.607, E3 +497097.198}
SPL {X  -137.967, Y  +286.821, Z    +0.000, E1   +43.969, E3 +497140.419}
ENDSPLINE

SPLINE
SPL {X  -149.143, Y  +306.414, Z    +0.000, E1   +36.361, E3 +497191.551}
SPL {X  -164.268, Y  +357.145, Z    +0.000, E1   +15.880, E3 +497149.311}
SPL {X  -165.510, Y  +371.680, Z    +0.000, E1    +7.684, E3 +497152.313}
SPL {X  -165.628, Y  +375.818, Z    +0.000, E1    +5.016, E3 +497160.242}
SPL {X  -165.650, Y  +383.362, Z    +0.000, E1    +0.177, E3 +497141.276}
SPL {X  -165.650, Y  +383.923, Z    +0.000, E1    -0.215, E3 +497154.433}
SPL {X  -165.650, Y  +388.083, Z    +0.000, E1    -3.355, E3 +497153.297}
SPL {X  -165.650, Y  +395.510, Z    +0.000, E1    -9.810, E3 +497149.423}
SPL {X  -165.650, Y  +403.066, Z    +0.000, E1   -17.886, E3 +497142.256}
SPL {X  -165.650, Y  +416.345, Z    +0.000, E1   -29.511, E3 +497143.999}
SPL {X  -165.650, Y  +422.331, Z    +0.000, E1   -27.760, E3 +497169.498}
SPL {X  -165.650, Y  +441.276, Z    +0.000, E1   -37.343, E3 +497179.355}
SPL {X  -165.650, Y  +462.890, Z    +0.000, E1   -40.484, E3 +497213.438}
ENDSPLINE

SPLINE
SPL {X  -165.650, Y  +446.920, Z    +0.000, E1   -31.238, E3 +497225.764}
ENDSPLINE

SPLINE
SPL {X  -165.650, Y  +447.935, Z    +0.000, E1   -30.213, E3 +497236.052}
SPL {X  -165.650, Y  +451.020, Z    +0.000, E1   -30.224, E3 +497246.872}
SPL {X  -165.650, Y  +454.519, Z    +0.000, E1   -30.374, E3 +497258.054}
SPL {X  -165.650, Y  +457.429, Z    +0.000, E1   -30.029, E3 +497270.756}
SPL {X  -165.650, Y  +461.678, Z    +0.000, E1   -30.426, E3 +497282.881}
SPL {X  -165.650, Y  +463.853, Z    +0.000, E1   -30.103, E3 +497292.720}
SPL {X  -165.650, Y  +468.397, Z    +0.000, E1   -30.302, E3 +497307.524}
SPL {X  -165.650, Y  +472.566, Z    +0.000, E1   -30.124, E3 +497323.234}
SPL {X  -165.650, Y  +475.265, Z    +0.000, E1   -30.034, E3 +497333.271}
SPL {X  -165.650, Y  +477.862, Z    +0.000, E1   -30.319, E3 +497340.463}
SPL {X  -165.650, Y  +481.042, Z    +0.000, E1   -30.192, E3 +497352.723}
SPL {X  -165.650, Y  +485.236, Z    +0.000, E1   -30.294, E3 +497366.578}
SPL {X  -165.650, Y  +488.041, Z    +0.000, E1   -30.253, E3 +497376.700}
SPL {X  -165.650, Y  +491.281, Z    +0.000, E1   -30.148, E3 +497388.838}
SPL {X  -165.650, Y  +495.051, Z    +0.000, E1   -30.213, E3 +497401.646}
SPL {X  -165.650, Y  +499.546, Z    +0.000, E1   -30.283, E3 +497417.089}
SPL {X  -165.650, Y  +503.544, Z    +0.000, E1   -30.247, E3 +497431.158}
SPL {X  -165.650, Y  +506.344, Z    +0.000, E1   -30.129, E3 +497441.826}
SPL {X  -165.650, Y  +510.660, Z    +0.000, E1   -30.223, E3 +497456.530}
SPL {X  -165.650, Y  +514.670, Z    +0.000, E1   -30.278, E3 +497470.040}
SPL {X  -165.650, Y  +517.919, Z    +0.000, E1   -30.227, E3 +497481.899}
SPL {X  -165.650, Y  +522.822, Z    +0.000, E1   -30.289, E3 +497498.788}
SPL {X  -165.650, Y  +527.393, Z    +0.000, E1   -30.104, E3 +497516.036}
SPL {X  -165.650, Y  +531.783, Z    +0.000, E1   -30.416, E3 +497529.214}
SPL {X  -165.650, Y  +534.115, Z    +0.000, E1   -30.089, E3 +497539.596}
SPL {X  -165.650, Y  +537.522, Z    +0.000, E1   -30.251, E3 +497550.510}
SPL {X  -165.650, Y  +540.621, Z    +0.000, E1   -30.014, E3 +497563.071}
SPL {X  -165.650, Y  +544.944, Z    +0.000, E1   -30.447, E3 +497575.271}
SPL {X  -165.650, Y  +547.199, Z    +0.000, E1   -30.132, E3 +497585.244}
SPL {X  -165.650, Y  +550.512, Z    +0.000, E1   -30.197, E3 +497596.570}
SPL {X  -165.650, Y  +553.852, Z    +0.000, E1   -30.156, E3 +497608.511}
SPL {X  -165.650, Y  +557.277, Z    +0.000, E1   -30.150, E3 +497620.685}
SPL {X  -165.650, Y  +561.168, Z    +0.000, E1   -30.194, E3 +497634.067}
SPL {X  -165.650, Y  +565.528, Z    +0.000, E1   -30.192, E3 +497649.550}
SPL {X  -165.650, Y  +570.048, Z    +0.000, E1   -30.238, E3 +497664.981}
SPL {X  -165.650, Y  +573.110, Z    +0.000, E1   -30.057, E3 +497676.966}
SPL {X  -165.650, Y  +577.587, Z    +0.000, E1   -30.270, E3 +497691.405}
SPL {X  -165.650, Y  +581.190, Z    +0.000, E1   -30.107, E3 +497705.044}
SPL {X  -165.650, Y  +585.053, Z    +0.000, E1   -30.090, E3 +497718.914}
ENDSPLINE

SPLINE
SPL {X  -165.650, Y  +484.445, Z    +0.000, E1   +32.277, E3 +497736.319}
SPL {X  -165.650, Y  +481.524, Z    +0.000, E1   +31.089, E3 +497753.769}
SPL {X  -165.650, Y  +478.014, Z    +0.000, E1   +30.826, E3 +497767.377}
SPL {X  -165.650, Y  +474.473, Z    +0.000, E1   +30.943, E3 +497778.701}
SPL {X  -165.650, Y  +471.826, Z    +0.000, E1   +30.770, E3 +497788.885}
SPL {X  -165.650, Y  +467.753, Z    +0.000, E1   +30.878, E3 +497802.258}
SPL {X  -165.650, Y  +463.837, Z    +0.000, E1   +30.924, E3 +497815.192}
SPL {X  -165.650, Y  +461.106, Z    +0.000, E1   +30.916, E3 +497824.579}
SPL {X  -165.650, Y  +457.156, Z    +0.000, E1   +30.860, E3 +497838.655}
SPL {X  -165.650, Y  +453.156, Z    +0.000, E1   +30.934, E3 +497851.629}
SPL {X  -165.650, Y  +450.433, Z    +0.000, E1   +30.789, E3 +497861.985}
SPL {X  -165.650, Y  +447.097, Z    +0.000, E1   +30.843, E3 +497873.033}
SPL {X  -165.650, Y  +443.673, Z    +0.000, E1   +30.907, E3 +497884.341}
SPL {X  -165.650, Y  +439.486, Z    +0.000, E1   +30.857, E3 +497899.150}
SPL {X  -165.650, Y  +435.146, Z    +0.000, E1   +30.969, E3 +497913.070}
SPL {X  -165.650, Y  +431.607, Z    +0.000, E1   +30.889, E3 +497925.784}
SPL {X  -165.650, Y  +427.340, Z    +0.000, E1   +30.870, E3 +497940.496}
SPL {X  -165.650, Y  +423.901, Z    +0.000, E1   +30.858, E3 +497952.252}
SPL {X  -165.650, Y  +421.437, Z    +0.000, E1   +30.833, E3 +497960.850}
SPL {X  -165.650, Y  +418.489, Z    +0.000, E1   +30.835, E3 +497970.967}
SPL {X  -165.650, Y  +414.127, Z    +0.000, E1   +30.869, E3 +497985.876}
SPL {X  -165.650, Y  +408.547, Z    +0.000, E1   +30.964, E3 +498004.291}
SPL {X  -165.650, Y  +405.433, Z    +0.000, E1   +30.730, E3 +498016.268}
SPL {X  -165.650, Y  +401.473, Z    +0.000, E1   +30.933, E3 +498028.717}
SPL {X  -165.650, Y  +396.018, Z    +0.000, E1   +30.861, E3 +498047.902}
SPL {X  -165.650, Y  +390.331, Z    +0.000, E1   +30.892, E3 +498067.154}
SPL {X  -165.650, Y  +384.849, Z    +0.000, E1   +30.885, E3 +498085.957}
SPL {X  -165.650, Y  +380.752, Z    +0.000, E1   +30.927, E3 +498099.459}
SPL {X  -165.648, Y  +377.739, Z    +0.000, E1   +30.835, E3 +498110.469}
SPL {X  -165.594, Y  +374.183, Z    +0.000, E1   +30.878, E3 +498122.305}
SPL {X  -165.492, Y  +371.263, Z    +0.000, E1   +30.913, E3 +498132.000}
SPL {X  -165.379, Y  +369.027, Z    +0.000, E1   +30.727, E3 +498140.939}
SPL {X  -165.167, Y  +365.866, Z    +0.000, E1   +30.741, E3 +498151.713}
SPL {X  -164.892, Y  +362.671, Z    +0.000, E1   +30.830, E3 +498162.037}
SPL {X  -164.570, Y  +359.612, Z    +0.000, E1   +30.773, E3 +498172.850}
SPL {X  -164.104, Y  +355.923, Z    +0.000, E1   +30.626, E3 +498186.566}
SPL {X  -163.573, Y  +352.353, Z    +0.000, E1   +30.451, E3 +498199.831}
SPL {X  -162.476, Y  +346.230, Z    +0.000, E1   +31.677, E3 +498212.412}
SPL {X  -152.976, Y  +314.952, Z    +0.000, E1   +38.607, E3 +498261.377}
SPL {X  -137.967, Y  +286.821, Z    +0.000, E1   +43.969, E3 +498304.598}
ENDSPLINE

SPLINE
SPL {X  -153.316, Y  +315.777, Z    +0.000, E1   +33.140, E3 +498347.226}
SPL {X  -164.446, Y  +358.564, Z    +0.000, E1   +15.149, E3 +498312.436}
SPL {X  -165.379, Y  +369.025, Z    +0.000, E1    +9.158, E3 +498318.161}
SPL {X  -165.612, Y  +374.969, Z    +0.000, E1    +5.630, E3 +498320.837}
SPL {X  -165.650, Y  +383.362, Z    +0.000, E1    +0.177, E3 +498305.455}
SPL {X  -165.650, Y  +383.923, Z    +0.000, E1    -0.215, E3 +498318.612}
SPL {X  -165.650, Y  +388.083, Z    +0.000, E1    -3.355, E3 +498317.476}
SPL {X  -165.650, Y  +393.983, Z    +0.000, E1    -8.501, E3 +498313.874}
SPL {X  -165.650, Y  +402.241, Z    +0.000, E1   -16.711, E3 +498308.386}
SPL {X  -165.650, Y  +416.345, Z    +0.000, E1   -29.511, E3 +498308.178}
SPL {X  -165.650, Y  +422.331, Z    +0.000, E1   -27.760, E3 +498333.677}
SPL {X  -165.650, Y  +441.276, Z    +0.000, E1   -37.343, E3 +498343.534}
SPL {X  -165.650, Y  +462.890, Z    +0.000, E1   -40.484, E3 +498377.617}
ENDSPLINE

SPLINE
SPL {X  -165.650, Y  +446.920, Z    +0.000, E1   -31.238, E3 +498389.943}
ENDSPLINE

SPLINE
SPL {X  -165.650, Y  +447.935, Z    +0.000, E1   -30.213, E3 +498400.231}
SPL {X  -165.650, Y  +451.020, Z    +0.000, E1   -30.224, E3 +498411.051}
SPL {X  -165.650, Y  +454.519, Z    +0.000, E1   -30.374, E3 +498422.233}
SPL {X  -165.650, Y  +457.429, Z    +0.000, E1   -30.029, E3 +498434.935}
SPL {X  -165.650, Y  +461.678, Z    +0.000, E1   -30.426, E3 +498447.060}
SPL {X  -165.650, Y  +463.853, Z    +0.000, E1   -30.103, E3 +498456.899}
SPL {X  -165.650, Y  +468.397, Z    +0.000, E1   -30.302, E3 +498471.703}
SPL {X  -165.650, Y  +472.566, Z    +0.000, E1   -30.124, E3 +498487.413}
SPL {X  -165.650, Y  +475.265, Z    +0.000, E1   -30.034, E3 +498497.450}
SPL {X  -165.650, Y  +479.559, Z    +0.000, E1   -30.258, E3 +498511.315}
SPL {X  -165.650, Y  +484.477, Z    +0.000, E1   -30.274, E3 +498528.324}
SPL {X  -165.650, Y  +489.057, Z    +0.000, E1   -30.341, E3 +498543.963}
SPL {X  -165.650, Y  +491.647, Z    +0.000, E1   -29.894, E3 +498555.897}
SPL {X  -165.650, Y  +495.051, Z    +0.000, E1   -30.213, E3 +498565.826}
SPL {X  -165.650, Y  +499.546, Z    +0.000, E1   -30.283, E3 +498581.268}
SPL {X  -165.650, Y  +503.544, Z    +0.000, E1   -30.247, E3 +498595.337}
SPL {X  -165.650, Y  +506.344, Z    +0.000, E1   -30.129, E3 +498606.006}
SPL {X  -165.650, Y  +510.660, Z    +0.000, E1   -30.223, E3 +498620.709}
SPL {X  -165.650, Y  +515.918, Z    +0.000, E1   -30.316, E3 +498638.517}
SPL {X  -165.650, Y  +520.621, Z    +0.000, E1   -30.198, E3 +498655.802}
SPL {X  -165.650, Y  +525.344, Z    +0.000, E1   -30.269, E3 +498671.859}
SPL {X  -165.650, Y  +528.152, Z    +0.000, E1   -29.991, E3 +498683.500}
SPL {X  -165.650, Y  +531.783, Z    +0.000, E1   -30.416, E3 +498693.393}
SPL {X  -165.650, Y  +534.115, Z    +0.000, E1   -30.089, E3 +498703.775}
SPL {X  -165.650, Y  +538.363, Z    +0.000, E1   -30.232, E3 +498717.945}
SPL {X  -165.650, Y  +543.650, Z    +0.000, E1   -30.281, E3 +498736.164}
SPL {X  -165.650, Y  +547.199, Z    +0.000, E1   -30.132, E3 +498749.423}
SPL {X  -165.650, Y  +550.512, Z    +0.000, E1   -30.197, E3 +498760.749}
SPL {X  -165.650, Y  +554.908, Z    +0.000, E1   -30.180, E3 +498776.410}
SPL {X  -165.650, Y  +560.243, Z    +0.000, E1   -30.214, E3 +498795.036}
SPL {X  -165.650, Y  +565.528, Z    +0.000, E1   -30.192, E3 +498813.729}
SPL {X  -165.650, Y  +570.048, Z    +0.000, E1   -30.238, E3 +498829.160}
SPL {X  -165.650, Y  +573.110, Z    +0.000, E1   -30.057, E3 +498841.145}
SPL {X  -165.650, Y  +577.587, Z    +0.000, E1   -30.270, E3 +498855.584}
SPL {X  -165.650, Y  +581.190, Z    +0.000, E1   -30.107, E3 +498869.223}
SPL {X  -165.650, Y  +585.053, Z    +0.000, E1   -30.090, E3 +498883.093}
ENDSPLINE

SPLINE
SPL {X  -165.650, Y  +484.968, Z    +0.000, E1   +32.508, E3 +498897.059}
SPL {X  -165.650, Y  +482.280, Z    +0.000, E1   +31.680, E3 +498911.386}
SPL {X  -165.650, Y  +479.331, Z    +0.000, E1   +30.680, E3 +498928.133}
SPL {X  -165.650, Y  +474.473, Z    +0.000, E1   +30.943, E3 +498942.880}
SPL {X  -165.650, Y  +470.376, Z    +0.000, E1   +30.888, E3 +498957.410}
SPL {X  -165.650, Y  +465.146, Z    +0.000, E1   +30.883, E3 +498975.340}
SPL {X  -165.650, Y  +461.106, Z    +0.000, E1   +30.916, E3 +498988.758}
SPL {X  -165.650, Y  +457.156, Z    +0.000, E1   +30.860, E3 +499002.835}
SPL {X  -165.650, Y  +453.156, Z    +0.000, E1   +30.934, E3 +499015.808}
SPL {X  -165.650, Y  +450.433, Z    +0.000, E1   +30.789, E3 +499026.164}
SPL {X  -165.650, Y  +447.097, Z    +0.000, E1   +30.843, E3 +499037.212}
SPL {X  -165.650, Y  +443.673, Z    +0.000, E1   +30.907, E3 +499048.520}
SPL {X  -165.650, Y  +439.486, Z    +0.000, E1   +30.857, E3 +499063.329}
SPL {X  -165.650, Y  +435.146, Z    +0.000, E1   +30.969, E3 +499077.249}
SPL {X  -165.650, Y  +431.607, Z    +0.000, E1   +30.889, E3 +499089.963}
SPL {X  -165.650, Y  +427.340, Z    +0.000, E1   +30.870, E3 +499104.675}
SPL {X  -165.650, Y  +423.901, Z    +0.000, E1   +30.858, E3 +499116.431}
SPL {X  -165.650, Y  +421.437, Z    +0.000, E1   +30.833, E3 +499125.029}
SPL {X  -165.650, Y  +418.489, Z    +0.000, E1   +30.835, E3 +499135.146}
SPL {X  -165.650, Y  +414.127, Z    +0.000, E1   +30.869, E3 +499150.055}
SPL {X  -165.650, Y  +408.547, Z    +0.000, E1   +30.964, E3 +499168.470}
SPL {X  -165.650, Y  +405.433, Z    +0.000, E1   +30.730, E3 +499180.447}
SPL {X  -165.650, Y  +402.516, Z    +0.000, E1   +30.874, E3 +499189.570}
SPL {X  -165.650, Y  +398.147, Z    +0.000, E1   +30.902, E3 +499204.449}
SPL {X  -165.650, Y  +394.694, Z    +0.000, E1   +30.805, E3 +499216.757}
SPL {X  -165.650, Y  +391.522, Z    +0.000, E1   +30.837, E3 +499227.438}
SPL {X  -165.650, Y  +387.533, Z    +0.000, E1   +30.858, E3 +499241.064}
SPL {X  -165.650, Y  +383.627, Z    +0.000, E1   +30.885, E3 +499254.124}
SPL {X  -165.650, Y  +379.886, Z    +0.000, E1   +30.887, E3 +499267.013}
SPL {X  -165.614, Y  +375.058, Z    +0.000, E1   +30.905, E3 +499283.466}
SPL {X  -165.492, Y  +371.263, Z    +0.000, E1   +30.913, E3 +499296.180}
SPL {X  -165.379, Y  +369.027, Z    +0.000, E1   +30.727, E3 +499305.118}
SPL {X  -165.167, Y  +365.866, Z    +0.000, E1   +30.741, E3 +499315.892}
SPL {X  -164.892, Y  +362.671, Z    +0.000, E1   +30.830, E3 +499326.216}
SPL {X  -164.570, Y  +359.612, Z    +0.000, E1   +30.773, E3 +499337.029}
SPL {X  -164.104, Y  +355.923, Z    +0.000, E1   +30.626, E3 +499350.745}
SPL {X  -163.573, Y  +352.353, Z    +0.000, E1   +30.451, E3 +499364.010}
SPL {X  -162.476, Y  +346.230, Z    +0.000, E1   +31.677, E3 +499376.591}
SPL {X  -152.976, Y  +314.952, Z    +0.000, E1   +38.607, E3 +499425.556}
SPL {X  -137.967, Y  +286.821, Z    +0.000, E1   +43.969, E3 +499468.777}
ENDSPLINE

SPLINE
SPL {X  -149.143, Y  +306.414, Z    +0.000, E1   +36.361, E3 +499519.910}
SPL {X  -163.091, Y  +349.496, Z    +0.000, E1   +19.699, E3 +499476.693}
SPL {X  -165.027, Y  +364.142, Z    +0.000, E1   +12.054, E3 +499479.833}
SPL {X  -165.612, Y  +374.969, Z    +0.000, E1    +5.630, E3 +499485.016}
SPL {X  -165.650, Y  +383.362, Z    +0.000, E1    +0.177, E3 +499469.634}
SPL {X  -165.650, Y  +383.923, Z    +0.000, E1    -0.215, E3 +499482.792}
SPL {X  -165.650, Y  +388.083, Z    +0.000, E1    -3.355, E3 +499481.655}
SPL {X  -165.650, Y  +393.983, Z    +0.000, E1    -8.501, E3 +499478.053}
SPL {X  -165.650, Y  +402.241, Z    +0.000, E1   -16.711, E3 +499472.565}
SPL {X  -165.650, Y  +414.811, Z    +0.000, E1   -28.314, E3 +499472.096}
SPL {X  -165.650, Y  +423.479, Z    +0.000, E1   -29.012, E3 +499496.024}
SPL {X  -165.650, Y  +441.276, Z    +0.000, E1   -37.343, E3 +499507.713}
SPL {X  -165.650, Y  +462.890, Z    +0.000, E1   -40.484, E3 +499541.796}
ENDSPLINE

SPLINE
SPL {X  -165.650, Y  +446.920, Z    +0.000, E1   -31.238, E3 +499554.122}
ENDSPLINE

SPLINE
SPL {X  -165.650, Y  +447.935, Z    +0.000, E1   -30.213, E3 +499564.410}
SPL {X  -165.650, Y  +451.020, Z    +0.000, E1   -30.224, E3 +499575.230}
SPL {X  -165.650, Y  +454.519, Z    +0.000, E1   -30.374, E3 +499586.413}
SPL {X  -165.650, Y  +456.542, Z    +0.000, E1   -29.986, E3 +499596.157}
SPL {X  -165.650, Y  +460.618, Z    +0.000, E1   -30.298, E3 +499608.478}
SPL {X  -165.650, Y  +463.853, Z    +0.000, E1   -30.103, E3 +499621.079}
SPL {X  -165.650, Y  +468.397, Z    +0.000, E1   -30.302, E3 +499635.882}
SPL {X  -165.650, Y  +472.566, Z    +0.000, E1   -30.124, E3 +499651.592}
SPL {X  -165.650, Y  +475.265, Z    +0.000, E1   -30.034, E3 +499661.629}
SPL {X  -165.650, Y  +479.559, Z    +0.000, E1   -30.258, E3 +499675.494}
SPL {X  -165.650, Y  +484.477, Z    +0.000, E1   -30.274, E3 +499692.503}
SPL {X  -165.650, Y  +488.041, Z    +0.000, E1   -30.253, E3 +499705.058}
SPL {X  -165.650, Y  +491.281, Z    +0.000, E1   -30.148, E3 +499717.196}
SPL {X  -165.650, Y  +495.051, Z    +0.000, E1   -30.213, E3 +499730.005}
SPL {X  -165.650, Y  +498.418, Z    +0.000, E1   -30.282, E3 +499741.298}
SPL {X  -165.650, Y  +502.421, Z    +0.000, E1   -30.263, E3 +499755.655}
SPL {X  -165.650, Y  +506.344, Z    +0.000, E1   -30.129, E3 +499770.185}
SPL {X  -165.650, Y  +509.866, Z    +0.000, E1   -30.236, E3 +499781.854}
SPL {X  -165.650, Y  +513.685, Z    +0.000, E1   -30.234, E3 +499795.350}
SPL {X  -165.650, Y  +517.919, Z    +0.000, E1   -30.227, E3 +499810.257}
SPL {X  -165.650, Y  +522.822, Z    +0.000, E1   -30.289, E3 +499827.146}
SPL {X  -165.650, Y  +527.393, Z    +0.000, E1   -30.104, E3 +499844.395}
SPL {X  -165.650, Y  +531.783, Z    +0.000, E1   -30.416, E3 +499857.572}
SPL {X  -165.650, Y  +534.115, Z    +0.000, E1   -30.089, E3 +499867.954}
SPL {X  -165.650, Y  +537.522, Z    +0.000, E1   -30.251, E3 +499878.868}
SPL {X  -165.650, Y  +540.621, Z    +0.000, E1   -30.014, E3 +499891.429}
SPL {X  -165.650, Y  +544.944, Z    +0.000, E1   -30.447, E3 +499903.629}
SPL {X  -165.650, Y  +548.549, Z    +0.000, E1   -30.216, E3 +499917.952}
SPL {X  -165.650, Y  +553.092, Z    +0.000, E1   -30.157, E3 +499934.295}
SPL {X  -165.650, Y  +556.274, Z    +0.000, E1   -30.127, E3 +499945.549}
SPL {X  -165.650, Y  +560.243, Z    +0.000, E1   -30.214, E3 +499959.215}
SPL {X  -165.650, Y  +565.528, Z    +0.000, E1   -30.192, E3 +499977.908}
SPL {X  -165.650, Y  +570.048, Z    +0.000, E1   -30.238, E3 +499993.339}
SPL {X  -165.650, Y  +573.110, Z    +0.000, E1   -30.057, E3 +500005.324}
SPL {X  -165.650, Y  +577.587, Z    +0.000, E1   -30.270, E3 +500019.763}
SPL {X  -165.650, Y  +581.190, Z    +0.000, E1   -30.107, E3 +500033.402}
SPL {X  -165.650, Y  +585.053, Z    +0.000, E1   -30.090, E3 +500047.272}
ENDSPLINE

